Universal Robots URScript: etalement.script

# UR5 - Protocole etalement cosmetique
# Genere automatiquement par ur5_etalement.py
# IMPORTANT : calibrer ROBOT_X_ORIGIN, ROBOT_Y_ORIGIN, ROBOT_Z_SURFACE avant execution
#
# === RECETTE DE REPRODUCTION ===
# Ce bloc enonce ce qui a produit ce fichier. Il ne porte pas de date :
# une date rendrait l export non reproductible, et git la porte deja.
# cycles : 6
#   cycle 1 : type=circular waypoints=200   label=Cycle 1 - Circulaire (UI)
#   cycle 2 : type=circular waypoints=200   label=Cycle 2 - Circulaire (UI)
#   cycle 3 : type=circular waypoints=200   label=Cycle 3 - Circulaire (UI)
#   cycle 4 : type=linear   waypoints=14    label=Cycle 4 - Triangulé (0deg)
#   cycle 5 : type=linear   waypoints=14    label=Cycle 5 - Triangulé (90deg)
#   cycle 6 : type=linear   waypoints=14    label=Cycle 6 - Triangulé (0deg)
# empreinte des reglages : 44136fa
#
# === PINCE 2F-85 : AUCUN ACTIONNEMENT ===
# Ce programme n a pas de commande de pince. La 2F-85 est un support
# passif pour le doigt silicone ; seule sa longueur (TCP_GRIPPER_Z=145 mm)
# entre dans set_tcp(). Aucun rq_activate / rq_* / RS485 outil / set_payload.
# Erreur PolyScope "wait for activation completed" au chargement = URCap
# Robotiq Grippers de l INSTALLATION du robot (auto-activation BeforeStart),
# pas ce fichier. Corriger sur le robot : Installation > URCaps/Gripper >
# desactiver l auto-activation, ou retirer le URCap, ou charger sur une
# installation sans pince.
#

# --- Ancre de la zone d'etalement ---
global P_REF = p[-0.011, 0.6, 0.05, 3.14159, 0.0, 0.0]

# --- Vitesses (m/s) par phase ---
# Note : URSCRIPT_MAX_TCP_SPEED (limite PolyScope, 0.25 m/s) n'est pas
# emis ici ; il est applique par le controleur. La vitesse de transit
# est inlinee directement sur les movel de transit.
global URSCRIPT_CONTACT_V = 0.0500  #sym:URSCRIPT_CONTACT_V
global URSCRIPT_RECONTACT_V = 0.0100  #sym:URSCRIPT_RECONTACT_V
global V_CIRC = 0.0360  #sym:CIRC_SPEED
global V_RECT = 0.0800  #sym:LIN_SPEED

# --- Accelerations (m/s^2) par phase ---
global URSCRIPT_ACCEL = 0.8  #sym:URSCRIPT_ACCEL
global A_INIT = 1.2  #sym:A_INIT

# --- Facteurs multiplicateurs globaux ---
global SPEED_FACTOR = 1.0
global ACCEL_FACTOR = 1.0
global URSCRIPT_BLEND = 0.002  #sym:URSCRIPT_BLEND

# --- Sondage de surface : 1 point en Z (sondage 3 points DESACTIVE, voir bloc commente) ---
global PROBE_FORCE_THR    = 4.0
global PROBE_DESCENT_V    = 0.0040
global PROBE_ACCEL        = 0.05
global PROBE_MAX_TRAVEL   = 0.15
global NOMINAL_FRAME = p[-0.011000, 0.592930, 0.050004, 3.141576, 0.000000, 0.000000]
global MEAS_FRAME = p[-0.011000, 0.592930, 0.050004, 3.141576, 0.000000, 0.000000]
global contact_found = False
global contact_pose = p[0,0,0,0,0,0]

# --- Sondage Z (1 point) : trouve le plan de la plaque par contact force ---
# Depart = pose courante (operateur jogge le doigt juste au-dessus du
# plateau). Descente en -Z (base) jusqu au contact ; le Z touche devient
# la reference de TOUS les cycles 1 a 6 via MEAS_FRAME.
def probe_surface_z():
  textmsg(">>> Sondage Z : 1 point (recherche du plateau)")
  start_pose = get_actual_tcp_pose()
  zero_ftsensor()
  sleep(0.2)
  # CB3 (PolyScope 3.x) : descente surveillee dans le thread principal
  # (speedl non bloquant + lecture force + stopl). Pas de thread (stopl/
  # movel interdits dans un thread). get_tcp_force() lu en entier, norme
  # calculee a la main (pas de slice [0:3], absent du parser CB3).
  f_norm = 0.0
  travel = 0.0
  while f_norm <= PROBE_FORCE_THR and travel < PROBE_MAX_TRAVEL:
    speedl([0, 0, -PROBE_DESCENT_V, 0, 0, 0], PROBE_ACCEL, 0.05)
    F_tcp = get_tcp_force()
    f_norm = sqrt(F_tcp[0]*F_tcp[0] + F_tcp[1]*F_tcp[1] + F_tcp[2]*F_tcp[2])
    cur = get_actual_tcp_pose()
    travel = start_pose[2] - cur[2]
  end
  stopl(2.0)
  if f_norm <= PROBE_FORCE_THR:
    popup("Sondage Z echoue - aucun contact", "Rapprocher le doigt du plateau puis relancer", error=True)
    halt
  end
  touch = get_actual_tcp_pose()
  # Reference Z des cycles : repere nominal translate en Z jusqu au plan
  # touche. Orientation/XY restent nominaux (1 point ne mesure pas
  # l inclinaison -> rework futur). apply_correction decale chaque
  # waypoint du meme dz ; force_mode(MEAS_FRAME) regule les 6 N en Z.
  MEAS_FRAME = p[NOMINAL_FRAME[0], NOMINAL_FRAME[1], touch[2], NOMINAL_FRAME[3], NOMINAL_FRAME[4], NOMINAL_FRAME[5]]
  textmsg("Plateau detecte, Z (m) = ", touch[2])
end

def apply_correction(p_world):
  return pose_trans(MEAS_FRAME, pose_trans(pose_inv(NOMINAL_FRAME), p_world))
end

def cycle_1():
  # --- Cycle 1 - Circulaire (UI) ---
  movel(apply_correction(p[-0.017788, 0.586142, 0.060004, 3.141576, 0.000000, 0.000000]), a=URSCRIPT_ACCEL*ACCEL_FACTOR, v=0.2500*SPEED_FACTOR)
  sleep(0.2)
  zero_ftsensor()
  sleep(0.2)
  force_mode(MEAS_FRAME, [0, 0, 1, 0, 0, 0], [0, 0, -6.0, 0, 0, 0], 2, [0.008, 0.008, 0.04, 0.35, 0.35, 0.35])
  movel(apply_correction(p[-0.017788, 0.586142, 0.045004, 3.141576, 0.000000, 0.000000]), a=URSCRIPT_ACCEL*ACCEL_FACTOR, v=URSCRIPT_RECONTACT_V*SPEED_FACTOR)
  movel(apply_correction(p[-0.017788, 0.586142, 0.050004, 3.141576, 0.000000, 0.000000]), a=URSCRIPT_ACCEL*ACCEL_FACTOR, v=V_CIRC*SPEED_FACTOR, r=URSCRIPT_BLEND)
  movel(apply_correction(p[-0.011098, 0.583533, 0.050004, 3.141576, 0.000000, 0.000000]), a=URSCRIPT_ACCEL*ACCEL_FACTOR, v=V_CIRC*SPEED_FACTOR, r=URSCRIPT_BLEND)
  movel(apply_correction(p[-0.004916, 0.587048, 0.050004, 3.141576, 0.000000, 0.000000]), a=URSCRIPT_ACCEL*ACCEL_FACTOR, v=V_CIRC*SPEED_FACTOR, r=URSCRIPT_BLEND)
  movel(apply_correction(p[-0.005086, 0.594004, 0.050004, 3.141576, 0.000000, 0.000000]), a=URSCRIPT_ACCEL*ACCEL_FACTOR, v=V_CIRC*SPEED_FACTOR, r=URSCRIPT_BLEND)
  movel(apply_correction(p[-0.011712, 0.596025, 0.050004, 3.141576, 0.000000, 0.000000]), a=URSCRIPT_ACCEL*ACCEL_FACTOR, v=V_CIRC*SPEED_FACTOR, r=URSCRIPT_BLEND)
  movel(apply_correction(p[-0.016472, 0.590781, 0.050004, 3.141576, 0.000000, 0.000000]), a=URSCRIPT_ACCEL*ACCEL_FACTOR, v=V_CIRC*SPEED_FACTOR, r=URSCRIPT_BLEND)
  movel(apply_correction(p[-0.015164, 0.583730, 0.050004, 3.141576, 0.000000, 0.000000]), a=URSCRIPT_ACCEL*ACCEL_FACTOR, v=V_CIRC*SPEED_FACTOR, r=URSCRIPT_BLEND)
  movel(apply_correction(p[-0.009065, 0.579930, 0.050004, 3.141576, 0.000000, 0.000000]), a=URSCRIPT_ACCEL*ACCEL_FACTOR, v=V_CIRC*SPEED_FACTOR, r=URSCRIPT_BLEND)
  movel(apply_correction(p[-0.002264, 0.582086, 0.050004, 3.141576, 0.000000, 0.000000]), a=URSCRIPT_ACCEL*ACCEL_FACTOR, v=V_CIRC*SPEED_FACTOR, r=URSCRIPT_BLEND)
  movel(apply_correction(p[-0.000623, 0.588885, 0.050004, 3.141576, 0.000000, 0.000000]), a=URSCRIPT_ACCEL*ACCEL_FACTOR, v=V_CIRC*SPEED_FACTOR, r=URSCRIPT_BLEND)
  movel(apply_correction(p[-0.006418, 0.592643, 0.050004, 3.141576, 0.000000, 0.000000]), a=URSCRIPT_ACCEL*ACCEL_FACTOR, v=V_CIRC*SPEED_FACTOR, r=URSCRIPT_BLEND)
  movel(apply_correction(p[-0.012226, 0.588648, 0.050004, 3.141576, 0.000000, 0.000000]), a=URSCRIPT_ACCEL*ACCEL_FACTOR, v=V_CIRC*SPEED_FACTOR, r=URSCRIPT_BLEND)
  movel(apply_correction(p[-0.012291, 0.581489, 0.050004, 3.141576, 0.000000, 0.000000]), a=URSCRIPT_ACCEL*ACCEL_FACTOR, v=V_CIRC*SPEED_FACTOR, r=URSCRIPT_BLEND)
  movel(apply_correction(p[-0.006988, 0.576638, 0.050004, 3.141576, 0.000000, 0.000000]), a=URSCRIPT_ACCEL*ACCEL_FACTOR, v=V_CIRC*SPEED_FACTOR, r=URSCRIPT_BLEND)
  movel(apply_correction(p[0.000125, 0.577386, 0.050004, 3.141576, 0.000000, 0.000000]), a=URSCRIPT_ACCEL*ACCEL_FACTOR, v=V_CIRC*SPEED_FACTOR, r=URSCRIPT_BLEND)
  movel(apply_correction(p[0.003408, 0.583603, 0.050004, 3.141576, 0.000000, 0.000000]), a=URSCRIPT_ACCEL*ACCEL_FACTOR, v=V_CIRC*SPEED_FACTOR, r=URSCRIPT_BLEND)
  movel(apply_correction(p[-0.001104, 0.588825, 0.050004, 3.141576, 0.000000, 0.000000]), a=URSCRIPT_ACCEL*ACCEL_FACTOR, v=V_CIRC*SPEED_FACTOR, r=URSCRIPT_BLEND)
  movel(apply_correction(p[-0.007670, 0.586361, 0.050004, 3.141576, 0.000000, 0.000000]), a=URSCRIPT_ACCEL*ACCEL_FACTOR, v=V_CIRC*SPEED_FACTOR, r=URSCRIPT_BLEND)
  movel(apply_correction(p[-0.009144, 0.579371, 0.050004, 3.141576, 0.000000, 0.000000]), a=URSCRIPT_ACCEL*ACCEL_FACTOR, v=V_CIRC*SPEED_FACTOR, r=URSCRIPT_BLEND)
  movel(apply_correction(p[-0.004813, 0.573634, 0.050004, 3.141576, 0.000000, 0.000000]), a=URSCRIPT_ACCEL*ACCEL_FACTOR, v=V_CIRC*SPEED_FACTOR, r=URSCRIPT_BLEND)
  movel(apply_correction(p[0.002324, 0.572985, 0.050004, 3.141576, 0.000000, 0.000000]), a=URSCRIPT_ACCEL*ACCEL_FACTOR, v=V_CIRC*SPEED_FACTOR, r=URSCRIPT_BLEND)
  movel(apply_correction(p[0.006999, 0.578286, 0.050004, 3.141576, 0.000000, 0.000000]), a=URSCRIPT_ACCEL*ACCEL_FACTOR, v=V_CIRC*SPEED_FACTOR, r=URSCRIPT_BLEND)
  movel(apply_correction(p[0.004110, 0.584567, 0.050004, 3.141576, 0.000000, 0.000000]), a=URSCRIPT_ACCEL*ACCEL_FACTOR, v=V_CIRC*SPEED_FACTOR, r=URSCRIPT_BLEND)
  movel(apply_correction(p[-0.002829, 0.583846, 0.050004, 3.141576, 0.000000, 0.000000]), a=URSCRIPT_ACCEL*ACCEL_FACTOR, v=V_CIRC*SPEED_FACTOR, r=URSCRIPT_BLEND)
  movel(apply_correction(p[-0.005691, 0.577324, 0.050004, 3.141576, 0.000000, 0.000000]), a=URSCRIPT_ACCEL*ACCEL_FACTOR, v=V_CIRC*SPEED_FACTOR, r=URSCRIPT_BLEND)
  movel(apply_correction(p[-0.002490, 0.570894, 0.050004, 3.141576, 0.000000, 0.000000]), a=URSCRIPT_ACCEL*ACCEL_FACTOR, v=V_CIRC*SPEED_FACTOR, r=URSCRIPT_BLEND)
  movel(apply_correction(p[0.004406, 0.568905, 0.050004, 3.141576, 0.000000, 0.000000]), a=URSCRIPT_ACCEL*ACCEL_FACTOR, v=V_CIRC*SPEED_FACTOR, r=URSCRIPT_BLEND)
  movel(apply_correction(p[0.010171, 0.573044, 0.050004, 3.141576, 0.000000, 0.000000]), a=URSCRIPT_ACCEL*ACCEL_FACTOR, v=V_CIRC*SPEED_FACTOR, r=URSCRIPT_BLEND)
  movel(apply_correction(p[0.009098, 0.579900, 0.050004, 3.141576, 0.000000, 0.000000]), a=URSCRIPT_ACCEL*ACCEL_FACTOR, v=V_CIRC*SPEED_FACTOR, r=URSCRIPT_BLEND)
  movel(apply_correction(p[0.002251, 0.581029, 0.050004, 3.141576, 0.000000, 0.000000]), a=URSCRIPT_ACCEL*ACCEL_FACTOR, v=V_CIRC*SPEED_FACTOR, r=URSCRIPT_BLEND)
  movel(apply_correction(p[-0.001925, 0.575290, 0.050004, 3.141576, 0.000000, 0.000000]), a=URSCRIPT_ACCEL*ACCEL_FACTOR, v=V_CIRC*SPEED_FACTOR, r=URSCRIPT_BLEND)
  movel(apply_correction(p[0.000027, 0.568386, 0.050004, 3.141576, 0.000000, 0.000000]), a=URSCRIPT_ACCEL*ACCEL_FACTOR, v=V_CIRC*SPEED_FACTOR, r=URSCRIPT_BLEND)
  movel(apply_correction(p[0.006439, 0.565146, 0.050005, 3.141576, 0.000000, 0.000000]), a=URSCRIPT_ACCEL*ACCEL_FACTOR, v=V_CIRC*SPEED_FACTOR, r=URSCRIPT_BLEND)
  movel(apply_correction(p[0.012978, 0.567972, 0.050004, 3.141576, 0.000000, 0.000000]), a=URSCRIPT_ACCEL*ACCEL_FACTOR, v=V_CIRC*SPEED_FACTOR, r=URSCRIPT_BLEND)
  movel(apply_correction(p[0.013753, 0.574903, 0.050004, 3.141576, 0.000000, 0.000000]), a=URSCRIPT_ACCEL*ACCEL_FACTOR, v=V_CIRC*SPEED_FACTOR, r=URSCRIPT_BLEND)
  movel(apply_correction(p[0.007496, 0.577845, 0.050004, 3.141576, 0.000000, 0.000000]), a=URSCRIPT_ACCEL*ACCEL_FACTOR, v=V_CIRC*SPEED_FACTOR, r=URSCRIPT_BLEND)
  movel(apply_correction(p[0.002166, 0.573206, 0.050004, 3.141576, 0.000000, 0.000000]), a=URSCRIPT_ACCEL*ACCEL_FACTOR, v=V_CIRC*SPEED_FACTOR, r=URSCRIPT_BLEND)
  movel(apply_correction(p[0.002775, 0.566066, 0.050004, 3.141576, 0.000000, 0.000000]), a=URSCRIPT_ACCEL*ACCEL_FACTOR, v=V_CIRC*SPEED_FACTOR, r=URSCRIPT_BLEND)
  movel(apply_correction(p[0.008487, 0.561706, 0.050005, 3.141576, 0.000000, 0.000000]), a=URSCRIPT_ACCEL*ACCEL_FACTOR, v=V_CIRC*SPEED_FACTOR, r=URSCRIPT_BLEND)
  movel(apply_correction(p[0.015475, 0.563167, 0.050005, 3.141576, 0.000000, 0.000000]), a=URSCRIPT_ACCEL*ACCEL_FACTOR, v=V_CIRC*SPEED_FACTOR, r=URSCRIPT_BLEND)
  movel(apply_correction(p[0.017743, 0.569730, 0.050004, 3.141576, 0.000000, 0.000000]), a=URSCRIPT_ACCEL*ACCEL_FACTOR, v=V_CIRC*SPEED_FACTOR, r=URSCRIPT_BLEND)
  movel(apply_correction(p[0.012260, 0.573881, 0.050004, 3.141576, 0.000000, 0.000000]), a=URSCRIPT_ACCEL*ACCEL_FACTOR, v=V_CIRC*SPEED_FACTOR, r=URSCRIPT_BLEND)
  movel(apply_correction(p[0.005935, 0.570677, 0.050004, 3.141576, 0.000000, 0.000000]), a=URSCRIPT_ACCEL*ACCEL_FACTOR, v=V_CIRC*SPEED_FACTOR, r=URSCRIPT_BLEND)
  movel(apply_correction(p[0.004428, 0.563644, 0.050005, 3.141576, 0.000000, 0.000000]), a=URSCRIPT_ACCEL*ACCEL_FACTOR, v=V_CIRC*SPEED_FACTOR, r=URSCRIPT_BLEND)
  movel(apply_correction(p[0.008552, 0.557768, 0.050005, 3.141576, 0.000000, 0.000000]), a=URSCRIPT_ACCEL*ACCEL_FACTOR, v=V_CIRC*SPEED_FACTOR, r=URSCRIPT_BLEND)
  movel(apply_correction(p[0.015598, 0.557554, 0.050005, 3.141576, 0.000000, 0.000000]), a=URSCRIPT_ACCEL*ACCEL_FACTOR, v=V_CIRC*SPEED_FACTOR, r=URSCRIPT_BLEND)
  movel(apply_correction(p[0.018398, 0.563819, 0.050005, 3.141576, 0.000000, 0.000000]), a=URSCRIPT_ACCEL*ACCEL_FACTOR, v=V_CIRC*SPEED_FACTOR, r=URSCRIPT_BLEND)
  movel(apply_correction(p[0.013349, 0.568656, 0.050004, 3.141576, 0.000000, 0.000000]), a=URSCRIPT_ACCEL*ACCEL_FACTOR, v=V_CIRC*SPEED_FACTOR, r=URSCRIPT_BLEND)
  movel(apply_correction(p[0.006365, 0.567164, 0.050004, 3.141576, 0.000000, 0.000000]), a=URSCRIPT_ACCEL*ACCEL_FACTOR, v=V_CIRC*SPEED_FACTOR, r=URSCRIPT_BLEND)
  movel(apply_correction(p[0.002726, 0.560986, 0.050005, 3.141576, 0.000000, 0.000000]), a=URSCRIPT_ACCEL*ACCEL_FACTOR, v=V_CIRC*SPEED_FACTOR, r=URSCRIPT_BLEND)
  movel(apply_correction(p[0.004975, 0.554229, 0.050005, 3.141576, 0.000000, 0.000000]), a=URSCRIPT_ACCEL*ACCEL_FACTOR, v=V_CIRC*SPEED_FACTOR, r=URSCRIPT_BLEND)
  movel(apply_correction(p[0.011813, 0.552992, 0.050005, 3.141576, 0.000000, 0.000000]), a=URSCRIPT_ACCEL*ACCEL_FACTOR, v=V_CIRC*SPEED_FACTOR, r=URSCRIPT_BLEND)
  movel(apply_correction(p[0.015059, 0.559096, 0.050005, 3.141576, 0.000000, 0.000000]), a=URSCRIPT_ACCEL*ACCEL_FACTOR, v=V_CIRC*SPEED_FACTOR, r=URSCRIPT_BLEND)
  movel(apply_correction(p[0.011046, 0.564958, 0.050005, 3.141576, 0.000000, 0.000000]), a=URSCRIPT_ACCEL*ACCEL_FACTOR, v=V_CIRC*SPEED_FACTOR, r=URSCRIPT_BLEND)
  movel(apply_correction(p[0.003896, 0.565651, 0.050004, 3.141576, 0.000000, 0.000000]), a=URSCRIPT_ACCEL*ACCEL_FACTOR, v=V_CIRC*SPEED_FACTOR, r=URSCRIPT_BLEND)
  movel(apply_correction(p[-0.001449, 0.560893, 0.050005, 3.141576, 0.000000, 0.000000]), a=URSCRIPT_ACCEL*ACCEL_FACTOR, v=V_CIRC*SPEED_FACTOR, r=URSCRIPT_BLEND)
  movel(apply_correction(p[-0.000730, 0.553895, 0.050005, 3.141576, 0.000000, 0.000000]), a=URSCRIPT_ACCEL*ACCEL_FACTOR, v=V_CIRC*SPEED_FACTOR, r=URSCRIPT_BLEND)
  movel(apply_correction(p[0.005938, 0.552136, 0.050005, 3.141576, 0.000000, 0.000000]), a=URSCRIPT_ACCEL*ACCEL_FACTOR, v=V_CIRC*SPEED_FACTOR, r=URSCRIPT_BLEND)
  movel(apply_correction(p[0.010014, 0.557869, 0.050005, 3.141576, 0.000000, 0.000000]), a=URSCRIPT_ACCEL*ACCEL_FACTOR, v=V_CIRC*SPEED_FACTOR, r=URSCRIPT_BLEND)
  movel(apply_correction(p[0.007718, 0.564641, 0.050005, 3.141576, 0.000000, 0.000000]), a=URSCRIPT_ACCEL*ACCEL_FACTOR, v=V_CIRC*SPEED_FACTOR, r=URSCRIPT_BLEND)
  movel(apply_correction(p[0.001166, 0.567570, 0.050004, 3.141576, 0.000000, 0.000000]), a=URSCRIPT_ACCEL*ACCEL_FACTOR, v=V_CIRC*SPEED_FACTOR, r=URSCRIPT_BLEND)
  movel(apply_correction(p[-0.005246, 0.564498, 0.050005, 3.141576, 0.000000, 0.000000]), a=URSCRIPT_ACCEL*ACCEL_FACTOR, v=V_CIRC*SPEED_FACTOR, r=URSCRIPT_BLEND)
  movel(apply_correction(p[-0.005654, 0.557540, 0.050005, 3.141576, 0.000000, 0.000000]), a=URSCRIPT_ACCEL*ACCEL_FACTOR, v=V_CIRC*SPEED_FACTOR, r=URSCRIPT_BLEND)
  movel(apply_correction(p[0.000763, 0.554955, 0.050005, 3.141576, 0.000000, 0.000000]), a=URSCRIPT_ACCEL*ACCEL_FACTOR, v=V_CIRC*SPEED_FACTOR, r=URSCRIPT_BLEND)
  movel(apply_correction(p[0.005879, 0.559839, 0.050005, 3.141576, 0.000000, 0.000000]), a=URSCRIPT_ACCEL*ACCEL_FACTOR, v=V_CIRC*SPEED_FACTOR, r=URSCRIPT_BLEND)
  movel(apply_correction(p[0.004993, 0.566952, 0.050004, 3.141576, 0.000000, 0.000000]), a=URSCRIPT_ACCEL*ACCEL_FACTOR, v=V_CIRC*SPEED_FACTOR, r=URSCRIPT_BLEND)
  movel(apply_correction(p[-0.000876, 0.571099, 0.050004, 3.141576, 0.000000, 0.000000]), a=URSCRIPT_ACCEL*ACCEL_FACTOR, v=V_CIRC*SPEED_FACTOR, r=URSCRIPT_BLEND)
  movel(apply_correction(p[-0.007807, 0.569384, 0.050004, 3.141576, 0.000000, 0.000000]), a=URSCRIPT_ACCEL*ACCEL_FACTOR, v=V_CIRC*SPEED_FACTOR, r=URSCRIPT_BLEND)
  movel(apply_correction(p[-0.009985, 0.562724, 0.050005, 3.141576, 0.000000, 0.000000]), a=URSCRIPT_ACCEL*ACCEL_FACTOR, v=V_CIRC*SPEED_FACTOR, r=URSCRIPT_BLEND)
  movel(apply_correction(p[-0.004550, 0.558471, 0.050005, 3.141576, 0.000000, 0.000000]), a=URSCRIPT_ACCEL*ACCEL_FACTOR, v=V_CIRC*SPEED_FACTOR, r=URSCRIPT_BLEND)
  movel(apply_correction(p[0.001532, 0.562013, 0.050005, 3.141576, 0.000000, 0.000000]), a=URSCRIPT_ACCEL*ACCEL_FACTOR, v=V_CIRC*SPEED_FACTOR, r=URSCRIPT_BLEND)
  movel(apply_correction(p[0.002038, 0.569150, 0.050004, 3.141576, 0.000000, 0.000000]), a=URSCRIPT_ACCEL*ACCEL_FACTOR, v=V_CIRC*SPEED_FACTOR, r=URSCRIPT_BLEND)
  movel(apply_correction(p[-0.002979, 0.574298, 0.050004, 3.141576, 0.000000, 0.000000]), a=URSCRIPT_ACCEL*ACCEL_FACTOR, v=V_CIRC*SPEED_FACTOR, r=URSCRIPT_BLEND)
  movel(apply_correction(p[-0.010128, 0.573991, 0.050004, 3.141576, 0.000000, 0.000000]), a=URSCRIPT_ACCEL*ACCEL_FACTOR, v=V_CIRC*SPEED_FACTOR, r=URSCRIPT_BLEND)
  movel(apply_correction(p[-0.013879, 0.568031, 0.050004, 3.141576, 0.000000, 0.000000]), a=URSCRIPT_ACCEL*ACCEL_FACTOR, v=V_CIRC*SPEED_FACTOR, r=URSCRIPT_BLEND)
  movel(apply_correction(p[-0.009845, 0.562427, 0.050005, 3.141576, 0.000000, 0.000000]), a=URSCRIPT_ACCEL*ACCEL_FACTOR, v=V_CIRC*SPEED_FACTOR, r=URSCRIPT_BLEND)
  movel(apply_correction(p[-0.003119, 0.564364, 0.050005, 3.141576, 0.000000, 0.000000]), a=URSCRIPT_ACCEL*ACCEL_FACTOR, v=V_CIRC*SPEED_FACTOR, r=URSCRIPT_BLEND)
  movel(apply_correction(p[-0.001202, 0.571240, 0.050004, 3.141576, 0.000000, 0.000000]), a=URSCRIPT_ACCEL*ACCEL_FACTOR, v=V_CIRC*SPEED_FACTOR, r=URSCRIPT_BLEND)
  movel(apply_correction(p[-0.005195, 0.577216, 0.050004, 3.141576, 0.000000, 0.000000]), a=URSCRIPT_ACCEL*ACCEL_FACTOR, v=V_CIRC*SPEED_FACTOR, r=URSCRIPT_BLEND)
  movel(apply_correction(p[-0.012283, 0.578294, 0.050004, 3.141576, 0.000000, 0.000000]), a=URSCRIPT_ACCEL*ACCEL_FACTOR, v=V_CIRC*SPEED_FACTOR, r=URSCRIPT_BLEND)
  movel(apply_correction(p[-0.017334, 0.573336, 0.050004, 3.141576, 0.000000, 0.000000]), a=URSCRIPT_ACCEL*ACCEL_FACTOR, v=V_CIRC*SPEED_FACTOR, r=URSCRIPT_BLEND)
  movel(apply_correction(p[-0.015002, 0.566819, 0.050004, 3.141576, 0.000000, 0.000000]), a=URSCRIPT_ACCEL*ACCEL_FACTOR, v=V_CIRC*SPEED_FACTOR, r=URSCRIPT_BLEND)
  movel(apply_correction(p[-0.008039, 0.566966, 0.050004, 3.141576, 0.000000, 0.000000]), a=URSCRIPT_ACCEL*ACCEL_FACTOR, v=V_CIRC*SPEED_FACTOR, r=URSCRIPT_BLEND)
  movel(apply_correction(p[-0.004752, 0.573277, 0.050004, 3.141576, 0.000000, 0.000000]), a=URSCRIPT_ACCEL*ACCEL_FACTOR, v=V_CIRC*SPEED_FACTOR, r=URSCRIPT_BLEND)
  movel(apply_correction(p[-0.007574, 0.579880, 0.050004, 3.141576, 0.000000, 0.000000]), a=URSCRIPT_ACCEL*ACCEL_FACTOR, v=V_CIRC*SPEED_FACTOR, r=URSCRIPT_BLEND)
  movel(apply_correction(p[-0.014343, 0.582272, 0.050004, 3.141576, 0.000000, 0.000000]), a=URSCRIPT_ACCEL*ACCEL_FACTOR, v=V_CIRC*SPEED_FACTOR, r=URSCRIPT_BLEND)
  movel(apply_correction(p[-0.020386, 0.578533, 0.050004, 3.141576, 0.000000, 0.000000]), a=URSCRIPT_ACCEL*ACCEL_FACTOR, v=V_CIRC*SPEED_FACTOR, r=URSCRIPT_BLEND)
  movel(apply_correction(p[-0.019895, 0.571600, 0.050004, 3.141576, 0.000000, 0.000000]), a=URSCRIPT_ACCEL*ACCEL_FACTOR, v=V_CIRC*SPEED_FACTOR, r=URSCRIPT_BLEND)
  movel(apply_correction(p[-0.013179, 0.569890, 0.050004, 3.141576, 0.000000, 0.000000]), a=URSCRIPT_ACCEL*ACCEL_FACTOR, v=V_CIRC*SPEED_FACTOR, r=URSCRIPT_BLEND)
  movel(apply_correction(p[-0.008631, 0.575334, 0.050004, 3.141576, 0.000000, 0.000000]), a=URSCRIPT_ACCEL*ACCEL_FACTOR, v=V_CIRC*SPEED_FACTOR, r=URSCRIPT_BLEND)
  movel(apply_correction(p[-0.010345, 0.582287, 0.050004, 3.141576, 0.000000, 0.000000]), a=URSCRIPT_ACCEL*ACCEL_FACTOR, v=V_CIRC*SPEED_FACTOR, r=URSCRIPT_BLEND)
  movel(apply_correction(p[-0.016696, 0.585620, 0.050004, 3.141576, 0.000000, 0.000000]), a=URSCRIPT_ACCEL*ACCEL_FACTOR, v=V_CIRC*SPEED_FACTOR, r=URSCRIPT_BLEND)
  movel(apply_correction(p[-0.023362, 0.583056, 0.050004, 3.141576, 0.000000, 0.000000]), a=URSCRIPT_ACCEL*ACCEL_FACTOR, v=V_CIRC*SPEED_FACTOR, r=URSCRIPT_BLEND)
  movel(apply_correction(p[-0.025236, 0.576243, 0.050004, 3.141576, 0.000000, 0.000000]), a=URSCRIPT_ACCEL*ACCEL_FACTOR, v=V_CIRC*SPEED_FACTOR, r=URSCRIPT_BLEND)
  movel(apply_correction(p[-0.020034, 0.571653, 0.050004, 3.141576, 0.000000, 0.000000]), a=URSCRIPT_ACCEL*ACCEL_FACTOR, v=V_CIRC*SPEED_FACTOR, r=URSCRIPT_BLEND)
  movel(apply_correction(p[-0.014038, 0.575090, 0.050004, 3.141576, 0.000000, 0.000000]), a=URSCRIPT_ACCEL*ACCEL_FACTOR, v=V_CIRC*SPEED_FACTOR, r=URSCRIPT_BLEND)
  movel(apply_correction(p[-0.014738, 0.582089, 0.050004, 3.141576, 0.000000, 0.000000]), a=URSCRIPT_ACCEL*ACCEL_FACTOR, v=V_CIRC*SPEED_FACTOR, r=URSCRIPT_BLEND)
  movel(apply_correction(p[-0.020976, 0.585534, 0.050004, 3.141576, 0.000000, 0.000000]), a=URSCRIPT_ACCEL*ACCEL_FACTOR, v=V_CIRC*SPEED_FACTOR, r=URSCRIPT_BLEND)
  movel(apply_correction(p[-0.027687, 0.583050, 0.050004, 3.141576, 0.000000, 0.000000]), a=URSCRIPT_ACCEL*ACCEL_FACTOR, v=V_CIRC*SPEED_FACTOR, r=URSCRIPT_BLEND)
  movel(apply_correction(p[-0.030305, 0.576399, 0.050004, 3.141576, 0.000000, 0.000000]), a=URSCRIPT_ACCEL*ACCEL_FACTOR, v=V_CIRC*SPEED_FACTOR, r=URSCRIPT_BLEND)
  movel(apply_correction(p[-0.026697, 0.570296, 0.050004, 3.141576, 0.000000, 0.000000]), a=URSCRIPT_ACCEL*ACCEL_FACTOR, v=V_CIRC*SPEED_FACTOR, r=URSCRIPT_BLEND)
  movel(apply_correction(p[-0.019718, 0.570534, 0.050004, 3.141576, 0.000000, 0.000000]), a=URSCRIPT_ACCEL*ACCEL_FACTOR, v=V_CIRC*SPEED_FACTOR, r=URSCRIPT_BLEND)
  movel(apply_correction(p[-0.017643, 0.577142, 0.050004, 3.141576, 0.000000, 0.000000]), a=URSCRIPT_ACCEL*ACCEL_FACTOR, v=V_CIRC*SPEED_FACTOR, r=URSCRIPT_BLEND)
  movel(apply_correction(p[-0.023092, 0.581572, 0.050004, 3.141576, 0.000000, 0.000000]), a=URSCRIPT_ACCEL*ACCEL_FACTOR, v=V_CIRC*SPEED_FACTOR, r=URSCRIPT_BLEND)
  movel(apply_correction(p[-0.029871, 0.579381, 0.050004, 3.141576, 0.000000, 0.000000]), a=URSCRIPT_ACCEL*ACCEL_FACTOR, v=V_CIRC*SPEED_FACTOR, r=URSCRIPT_BLEND)
  movel(apply_correction(p[-0.032536, 0.572708, 0.050004, 3.141576, 0.000000, 0.000000]), a=URSCRIPT_ACCEL*ACCEL_FACTOR, v=V_CIRC*SPEED_FACTOR, r=URSCRIPT_BLEND)
  movel(apply_correction(p[-0.029339, 0.566277, 0.050004, 3.141576, 0.000000, 0.000000]), a=URSCRIPT_ACCEL*ACCEL_FACTOR, v=V_CIRC*SPEED_FACTOR, r=URSCRIPT_BLEND)
  movel(apply_correction(p[-0.022399, 0.564726, 0.050005, 3.141576, 0.000000, 0.000000]), a=URSCRIPT_ACCEL*ACCEL_FACTOR, v=V_CIRC*SPEED_FACTOR, r=URSCRIPT_BLEND)
  movel(apply_correction(p[-0.017535, 0.569747, 0.050004, 3.141576, 0.000000, 0.000000]), a=URSCRIPT_ACCEL*ACCEL_FACTOR, v=V_CIRC*SPEED_FACTOR, r=URSCRIPT_BLEND)
  movel(apply_correction(p[-0.020477, 0.575989, 0.050004, 3.141576, 0.000000, 0.000000]), a=URSCRIPT_ACCEL*ACCEL_FACTOR, v=V_CIRC*SPEED_FACTOR, r=URSCRIPT_BLEND)
  movel(apply_correction(p[-0.027450, 0.575397, 0.050004, 3.141576, 0.000000, 0.000000]), a=URSCRIPT_ACCEL*ACCEL_FACTOR, v=V_CIRC*SPEED_FACTOR, r=URSCRIPT_BLEND)
  movel(apply_correction(p[-0.030496, 0.568956, 0.050004, 3.141576, 0.000000, 0.000000]), a=URSCRIPT_ACCEL*ACCEL_FACTOR, v=V_CIRC*SPEED_FACTOR, r=URSCRIPT_BLEND)
  movel(apply_correction(p[-0.027445, 0.562453, 0.050005, 3.141576, 0.000000, 0.000000]), a=URSCRIPT_ACCEL*ACCEL_FACTOR, v=V_CIRC*SPEED_FACTOR, r=URSCRIPT_BLEND)
  movel(apply_correction(p[-0.020600, 0.560297, 0.050005, 3.141576, 0.000000, 0.000000]), a=URSCRIPT_ACCEL*ACCEL_FACTOR, v=V_CIRC*SPEED_FACTOR, r=URSCRIPT_BLEND)
  movel(apply_correction(p[-0.014717, 0.564274, 0.050005, 3.141576, 0.000000, 0.000000]), a=URSCRIPT_ACCEL*ACCEL_FACTOR, v=V_CIRC*SPEED_FACTOR, r=URSCRIPT_BLEND)
  movel(apply_correction(p[-0.015552, 0.571170, 0.050004, 3.141576, 0.000000, 0.000000]), a=URSCRIPT_ACCEL*ACCEL_FACTOR, v=V_CIRC*SPEED_FACTOR, r=URSCRIPT_BLEND)
  movel(apply_correction(p[-0.022352, 0.572534, 0.050004, 3.141576, 0.000000, 0.000000]), a=URSCRIPT_ACCEL*ACCEL_FACTOR, v=V_CIRC*SPEED_FACTOR, r=URSCRIPT_BLEND)
  movel(apply_correction(p[-0.026686, 0.566919, 0.050004, 3.141576, 0.000000, 0.000000]), a=URSCRIPT_ACCEL*ACCEL_FACTOR, v=V_CIRC*SPEED_FACTOR, r=URSCRIPT_BLEND)
  movel(apply_correction(p[-0.024903, 0.559969, 0.050005, 3.141576, 0.000000, 0.000000]), a=URSCRIPT_ACCEL*ACCEL_FACTOR, v=V_CIRC*SPEED_FACTOR, r=URSCRIPT_BLEND)
  movel(apply_correction(p[-0.018568, 0.556581, 0.050005, 3.141576, 0.000000, 0.000000]), a=URSCRIPT_ACCEL*ACCEL_FACTOR, v=V_CIRC*SPEED_FACTOR, r=URSCRIPT_BLEND)
  movel(apply_correction(p[-0.011952, 0.559230, 0.050005, 3.141576, 0.000000, 0.000000]), a=URSCRIPT_ACCEL*ACCEL_FACTOR, v=V_CIRC*SPEED_FACTOR, r=URSCRIPT_BLEND)
  movel(apply_correction(p[-0.010947, 0.566137, 0.050004, 3.141576, 0.000000, 0.000000]), a=URSCRIPT_ACCEL*ACCEL_FACTOR, v=V_CIRC*SPEED_FACTOR, r=URSCRIPT_BLEND)
  movel(apply_correction(p[-0.017092, 0.569298, 0.050004, 3.141576, 0.000000, 0.000000]), a=URSCRIPT_ACCEL*ACCEL_FACTOR, v=V_CIRC*SPEED_FACTOR, r=URSCRIPT_BLEND)
  movel(apply_correction(p[-0.022556, 0.564825, 0.050005, 3.141576, 0.000000, 0.000000]), a=URSCRIPT_ACCEL*ACCEL_FACTOR, v=V_CIRC*SPEED_FACTOR, r=URSCRIPT_BLEND)
  movel(apply_correction(p[-0.022123, 0.557672, 0.050005, 3.141576, 0.000000, 0.000000]), a=URSCRIPT_ACCEL*ACCEL_FACTOR, v=V_CIRC*SPEED_FACTOR, r=URSCRIPT_BLEND)
  movel(apply_correction(p[-0.016514, 0.553178, 0.050005, 3.141576, 0.000000, 0.000000]), a=URSCRIPT_ACCEL*ACCEL_FACTOR, v=V_CIRC*SPEED_FACTOR, r=URSCRIPT_BLEND)
  movel(apply_correction(p[-0.009477, 0.554429, 0.050005, 3.141576, 0.000000, 0.000000]), a=URSCRIPT_ACCEL*ACCEL_FACTOR, v=V_CIRC*SPEED_FACTOR, r=URSCRIPT_BLEND)
  movel(apply_correction(p[-0.006757, 0.560900, 0.050005, 3.141576, 0.000000, 0.000000]), a=URSCRIPT_ACCEL*ACCEL_FACTOR, v=V_CIRC*SPEED_FACTOR, r=URSCRIPT_BLEND)
  movel(apply_correction(p[-0.011771, 0.565641, 0.050004, 3.141576, 0.000000, 0.000000]), a=URSCRIPT_ACCEL*ACCEL_FACTOR, v=V_CIRC*SPEED_FACTOR, r=URSCRIPT_BLEND)
  movel(apply_correction(p[-0.018106, 0.562599, 0.050005, 3.141576, 0.000000, 0.000000]), a=URSCRIPT_ACCEL*ACCEL_FACTOR, v=V_CIRC*SPEED_FACTOR, r=URSCRIPT_BLEND)
  movel(apply_correction(p[-0.019075, 0.555515, 0.050005, 3.141576, 0.000000, 0.000000]), a=URSCRIPT_ACCEL*ACCEL_FACTOR, v=V_CIRC*SPEED_FACTOR, r=URSCRIPT_BLEND)
  movel(apply_correction(p[-0.014379, 0.550076, 0.050005, 3.141576, 0.000000, 0.000000]), a=URSCRIPT_ACCEL*ACCEL_FACTOR, v=V_CIRC*SPEED_FACTOR, r=URSCRIPT_BLEND)
  movel(apply_correction(p[-0.007220, 0.549921, 0.050005, 3.141576, 0.000000, 0.000000]), a=URSCRIPT_ACCEL*ACCEL_FACTOR, v=V_CIRC*SPEED_FACTOR, r=URSCRIPT_BLEND)
  movel(apply_correction(p[-0.003008, 0.555581, 0.050005, 3.141576, 0.000000, 0.000000]), a=URSCRIPT_ACCEL*ACCEL_FACTOR, v=V_CIRC*SPEED_FACTOR, r=URSCRIPT_BLEND)
  movel(apply_correction(p[-0.006508, 0.561538, 0.050005, 3.141576, 0.000000, 0.000000]), a=URSCRIPT_ACCEL*ACCEL_FACTOR, v=V_CIRC*SPEED_FACTOR, r=URSCRIPT_BLEND)
  movel(apply_correction(p[-0.013362, 0.560174, 0.050005, 3.141576, 0.000000, 0.000000]), a=URSCRIPT_ACCEL*ACCEL_FACTOR, v=V_CIRC*SPEED_FACTOR, r=URSCRIPT_BLEND)
  movel(apply_correction(p[-0.015736, 0.553449, 0.050005, 3.141576, 0.000000, 0.000000]), a=URSCRIPT_ACCEL*ACCEL_FACTOR, v=V_CIRC*SPEED_FACTOR, r=URSCRIPT_BLEND)
  movel(apply_correction(p[-0.012114, 0.547244, 0.050005, 3.141576, 0.000000, 0.000000]), a=URSCRIPT_ACCEL*ACCEL_FACTOR, v=V_CIRC*SPEED_FACTOR, r=URSCRIPT_BLEND)
  movel(apply_correction(p[-0.005103, 0.545724, 0.050005, 3.141576, 0.000000, 0.000000]), a=URSCRIPT_ACCEL*ACCEL_FACTOR, v=V_CIRC*SPEED_FACTOR, r=URSCRIPT_BLEND)
  movel(apply_correction(p[0.000267, 0.550317, 0.050005, 3.141576, 0.000000, 0.000000]), a=URSCRIPT_ACCEL*ACCEL_FACTOR, v=V_CIRC*SPEED_FACTOR, r=URSCRIPT_BLEND)
  movel(apply_correction(p[-0.001550, 0.556944, 0.050005, 3.141576, 0.000000, 0.000000]), a=URSCRIPT_ACCEL*ACCEL_FACTOR, v=V_CIRC*SPEED_FACTOR, r=URSCRIPT_BLEND)
  movel(apply_correction(p[-0.008498, 0.557307, 0.050005, 3.141576, 0.000000, 0.000000]), a=URSCRIPT_ACCEL*ACCEL_FACTOR, v=V_CIRC*SPEED_FACTOR, r=URSCRIPT_BLEND)
  movel(apply_correction(p[-0.012498, 0.551407, 0.050005, 3.141576, 0.000000, 0.000000]), a=URSCRIPT_ACCEL*ACCEL_FACTOR, v=V_CIRC*SPEED_FACTOR, r=URSCRIPT_BLEND)
  movel(apply_correction(p[-0.010765, 0.544449, 0.050005, 3.141576, 0.000000, 0.000000]), a=URSCRIPT_ACCEL*ACCEL_FACTOR, v=V_CIRC*SPEED_FACTOR, r=URSCRIPT_BLEND)
  movel(apply_correction(p[-0.004471, 0.541100, 0.050005, 3.141576, 0.000000, 0.000000]), a=URSCRIPT_ACCEL*ACCEL_FACTOR, v=V_CIRC*SPEED_FACTOR, r=URSCRIPT_BLEND)
  movel(apply_correction(p[0.001548, 0.544594, 0.050005, 3.141576, 0.000000, 0.000000]), a=URSCRIPT_ACCEL*ACCEL_FACTOR, v=V_CIRC*SPEED_FACTOR, r=URSCRIPT_BLEND)
  movel(apply_correction(p[0.000165, 0.551320, 0.050005, 3.141576, 0.000000, 0.000000]), a=URSCRIPT_ACCEL*ACCEL_FACTOR, v=V_CIRC*SPEED_FACTOR, r=URSCRIPT_BLEND)
  movel(apply_correction(p[-0.006728, 0.552924, 0.050005, 3.141576, 0.000000, 0.000000]), a=URSCRIPT_ACCEL*ACCEL_FACTOR, v=V_CIRC*SPEED_FACTOR, r=URSCRIPT_BLEND)
  movel(apply_correction(p[-0.012333, 0.548421, 0.050005, 3.141576, 0.000000, 0.000000]), a=URSCRIPT_ACCEL*ACCEL_FACTOR, v=V_CIRC*SPEED_FACTOR, r=URSCRIPT_BLEND)
  movel(apply_correction(p[-0.012858, 0.541260, 0.050005, 3.141576, 0.000000, 0.000000]), a=URSCRIPT_ACCEL*ACCEL_FACTOR, v=V_CIRC*SPEED_FACTOR, r=URSCRIPT_BLEND)
  movel(apply_correction(p[-0.007599, 0.536545, 0.050005, 3.141576, 0.000000, 0.000000]), a=URSCRIPT_ACCEL*ACCEL_FACTOR, v=V_CIRC*SPEED_FACTOR, r=URSCRIPT_BLEND)
  movel(apply_correction(p[-0.001356, 0.539401, 0.050005, 3.141576, 0.000000, 0.000000]), a=URSCRIPT_ACCEL*ACCEL_FACTOR, v=V_CIRC*SPEED_FACTOR, r=URSCRIPT_BLEND)
  movel(apply_correction(p[-0.002041, 0.546340, 0.050005, 3.141576, 0.000000, 0.000000]), a=URSCRIPT_ACCEL*ACCEL_FACTOR, v=V_CIRC*SPEED_FACTOR, r=URSCRIPT_BLEND)
  movel(apply_correction(p[-0.008378, 0.549617, 0.050005, 3.141576, 0.000000, 0.000000]), a=URSCRIPT_ACCEL*ACCEL_FACTOR, v=V_CIRC*SPEED_FACTOR, r=URSCRIPT_BLEND)
  movel(apply_correction(p[-0.015100, 0.547118, 0.050005, 3.141576, 0.000000, 0.000000]), a=URSCRIPT_ACCEL*ACCEL_FACTOR, v=V_CIRC*SPEED_FACTOR, r=URSCRIPT_BLEND)
  movel(apply_correction(p[-0.017677, 0.540470, 0.050005, 3.141576, 0.000000, 0.000000]), a=URSCRIPT_ACCEL*ACCEL_FACTOR, v=V_CIRC*SPEED_FACTOR, r=URSCRIPT_BLEND)
  movel(apply_correction(p[-0.013312, 0.535048, 0.050005, 3.141576, 0.000000, 0.000000]), a=URSCRIPT_ACCEL*ACCEL_FACTOR, v=V_CIRC*SPEED_FACTOR, r=URSCRIPT_BLEND)
  movel(apply_correction(p[-0.006869, 0.537498, 0.050005, 3.141576, 0.000000, 0.000000]), a=URSCRIPT_ACCEL*ACCEL_FACTOR, v=V_CIRC*SPEED_FACTOR, r=URSCRIPT_BLEND)
  movel(apply_correction(p[-0.006196, 0.544557, 0.050005, 3.141576, 0.000000, 0.000000]), a=URSCRIPT_ACCEL*ACCEL_FACTOR, v=V_CIRC*SPEED_FACTOR, r=URSCRIPT_BLEND)
  movel(apply_correction(p[-0.011303, 0.549604, 0.050005, 3.141576, 0.000000, 0.000000]), a=URSCRIPT_ACCEL*ACCEL_FACTOR, v=V_CIRC*SPEED_FACTOR, r=URSCRIPT_BLEND)
  movel(apply_correction(p[-0.018457, 0.549307, 0.050005, 3.141576, 0.000000, 0.000000]), a=URSCRIPT_ACCEL*ACCEL_FACTOR, v=V_CIRC*SPEED_FACTOR, r=URSCRIPT_BLEND)
  movel(apply_correction(p[-0.022436, 0.543491, 0.050005, 3.141576, 0.000000, 0.000000]), a=URSCRIPT_ACCEL*ACCEL_FACTOR, v=V_CIRC*SPEED_FACTOR, r=URSCRIPT_BLEND)
  movel(apply_correction(p[-0.018669, 0.537715, 0.050005, 3.141576, 0.000000, 0.000000]), a=URSCRIPT_ACCEL*ACCEL_FACTOR, v=V_CIRC*SPEED_FACTOR, r=URSCRIPT_BLEND)
  movel(apply_correction(p[-0.011875, 0.539380, 0.050005, 3.141576, 0.000000, 0.000000]), a=URSCRIPT_ACCEL*ACCEL_FACTOR, v=V_CIRC*SPEED_FACTOR, r=URSCRIPT_BLEND)
  movel(apply_correction(p[-0.009742, 0.546188, 0.050005, 3.141576, 0.000000, 0.000000]), a=URSCRIPT_ACCEL*ACCEL_FACTOR, v=V_CIRC*SPEED_FACTOR, r=URSCRIPT_BLEND)
  movel(apply_correction(p[-0.013558, 0.552276, 0.050005, 3.141576, 0.000000, 0.000000]), a=URSCRIPT_ACCEL*ACCEL_FACTOR, v=V_CIRC*SPEED_FACTOR, r=URSCRIPT_BLEND)
  movel(apply_correction(p[-0.020613, 0.553566, 0.050005, 3.141576, 0.000000, 0.000000]), a=URSCRIPT_ACCEL*ACCEL_FACTOR, v=V_CIRC*SPEED_FACTOR, r=URSCRIPT_BLEND)
  movel(apply_correction(p[-0.025840, 0.548787, 0.050005, 3.141576, 0.000000, 0.000000]), a=URSCRIPT_ACCEL*ACCEL_FACTOR, v=V_CIRC*SPEED_FACTOR, r=URSCRIPT_BLEND)
  movel(apply_correction(p[-0.023792, 0.542172, 0.050005, 3.141576, 0.000000, 0.000000]), a=URSCRIPT_ACCEL*ACCEL_FACTOR, v=V_CIRC*SPEED_FACTOR, r=URSCRIPT_BLEND)
  movel(apply_correction(p[-0.016835, 0.542028, 0.050005, 3.141576, 0.000000, 0.000000]), a=URSCRIPT_ACCEL*ACCEL_FACTOR, v=V_CIRC*SPEED_FACTOR, r=URSCRIPT_BLEND)
  movel(apply_correction(p[-0.013339, 0.548221, 0.050005, 3.141576, 0.000000, 0.000000]), a=URSCRIPT_ACCEL*ACCEL_FACTOR, v=V_CIRC*SPEED_FACTOR, r=URSCRIPT_BLEND)
  movel(apply_correction(p[-0.015968, 0.554903, 0.050005, 3.141576, 0.000000, 0.000000]), a=URSCRIPT_ACCEL*ACCEL_FACTOR, v=V_CIRC*SPEED_FACTOR, r=URSCRIPT_BLEND)
  movel(apply_correction(p[-0.022664, 0.557493, 0.050005, 3.141576, 0.000000, 0.000000]), a=URSCRIPT_ACCEL*ACCEL_FACTOR, v=V_CIRC*SPEED_FACTOR, r=URSCRIPT_BLEND)
  movel(apply_correction(p[-0.028833, 0.553959, 0.050005, 3.141576, 0.000000, 0.000000]), a=URSCRIPT_ACCEL*ACCEL_FACTOR, v=V_CIRC*SPEED_FACTOR, r=URSCRIPT_BLEND)
  movel(apply_correction(p[-0.028635, 0.547007, 0.050005, 3.141576, 0.000000, 0.000000]), a=URSCRIPT_ACCEL*ACCEL_FACTOR, v=V_CIRC*SPEED_FACTOR, r=URSCRIPT_BLEND)
  movel(apply_correction(p[-0.022003, 0.545011, 0.050005, 3.141576, 0.000000, 0.000000]), a=URSCRIPT_ACCEL*ACCEL_FACTOR, v=V_CIRC*SPEED_FACTOR, r=URSCRIPT_BLEND)
  movel(apply_correction(p[-0.017259, 0.550270, 0.050005, 3.141576, 0.000000, 0.000000]), a=URSCRIPT_ACCEL*ACCEL_FACTOR, v=V_CIRC*SPEED_FACTOR, r=URSCRIPT_BLEND)
  movel(apply_correction(p[-0.018587, 0.557319, 0.050005, 3.141576, 0.000000, 0.000000]), a=URSCRIPT_ACCEL*ACCEL_FACTOR, v=V_CIRC*SPEED_FACTOR, r=URSCRIPT_BLEND)
  movel(apply_correction(p[-0.024697, 0.561102, 0.050005, 3.141576, 0.000000, 0.000000]), a=URSCRIPT_ACCEL*ACCEL_FACTOR, v=V_CIRC*SPEED_FACTOR, r=URSCRIPT_BLEND)
  movel(apply_correction(p[-0.031491, 0.558927, 0.050005, 3.141576, 0.000000, 0.000000]), a=URSCRIPT_ACCEL*ACCEL_FACTOR, v=V_CIRC*SPEED_FACTOR, r=URSCRIPT_BLEND)
  movel(apply_correction(p[-0.033105, 0.552122, 0.050005, 3.141576, 0.000000, 0.000000]), a=URSCRIPT_ACCEL*ACCEL_FACTOR, v=V_CIRC*SPEED_FACTOR, r=URSCRIPT_BLEND)
  movel(apply_correction(p[-0.027295, 0.548386, 0.050005, 3.141576, 0.000000, 0.000000]), a=URSCRIPT_ACCEL*ACCEL_FACTOR, v=V_CIRC*SPEED_FACTOR, r=URSCRIPT_BLEND)
  movel(apply_correction(p[-0.021500, 0.552402, 0.050005, 3.141576, 0.000000, 0.000000]), a=URSCRIPT_ACCEL*ACCEL_FACTOR, v=V_CIRC*SPEED_FACTOR, r=URSCRIPT_BLEND)
  movel(apply_correction(p[-0.021456, 0.559562, 0.050005, 3.141576, 0.000000, 0.000000]), a=URSCRIPT_ACCEL*ACCEL_FACTOR, v=V_CIRC*SPEED_FACTOR, r=URSCRIPT_BLEND)
  movel(apply_correction(p[-0.026772, 0.564399, 0.050005, 3.141576, 0.000000, 0.000000]), a=URSCRIPT_ACCEL*ACCEL_FACTOR, v=V_CIRC*SPEED_FACTOR, r=URSCRIPT_BLEND)
  movel(apply_correction(p[-0.033883, 0.563631, 0.050005, 3.141576, 0.000000, 0.000000]), a=URSCRIPT_ACCEL*ACCEL_FACTOR, v=V_CIRC*SPEED_FACTOR, r=URSCRIPT_BLEND)
  movel(apply_correction(p[-0.037145, 0.557401, 0.050005, 3.141576, 0.000000, 0.000000]), a=URSCRIPT_ACCEL*ACCEL_FACTOR, v=V_CIRC*SPEED_FACTOR, r=URSCRIPT_BLEND)
  movel(apply_correction(p[-0.032611, 0.552198, 0.050005, 3.141576, 0.000000, 0.000000]), a=URSCRIPT_ACCEL*ACCEL_FACTOR, v=V_CIRC*SPEED_FACTOR, r=URSCRIPT_BLEND)
  movel(apply_correction(p[-0.026054, 0.554687, 0.050005, 3.141576, 0.000000, 0.000000]), a=URSCRIPT_ACCEL*ACCEL_FACTOR, v=V_CIRC*SPEED_FACTOR, r=URSCRIPT_BLEND)
  movel(apply_correction(p[-0.024601, 0.561681, 0.050005, 3.141576, 0.000000, 0.000000]), a=URSCRIPT_ACCEL*ACCEL_FACTOR, v=V_CIRC*SPEED_FACTOR, r=URSCRIPT_BLEND)
  movel(apply_correction(p[-0.028946, 0.567405, 0.050004, 3.141576, 0.000000, 0.000000]), a=URSCRIPT_ACCEL*ACCEL_FACTOR, v=V_CIRC*SPEED_FACTOR, r=URSCRIPT_BLEND)
  movel(apply_correction(p[-0.036085, 0.568036, 0.050004, 3.141576, 0.000000, 0.000000]), a=URSCRIPT_ACCEL*ACCEL_FACTOR, v=V_CIRC*SPEED_FACTOR, r=URSCRIPT_BLEND)
  movel(apply_correction(p[-0.040740, 0.562720, 0.050005, 3.141576, 0.000000, 0.000000]), a=URSCRIPT_ACCEL*ACCEL_FACTOR, v=V_CIRC*SPEED_FACTOR, r=URSCRIPT_BLEND)
  movel(apply_correction(p[-0.037827, 0.556450, 0.050005, 3.141576, 0.000000, 0.000000]), a=URSCRIPT_ACCEL*ACCEL_FACTOR, v=V_CIRC*SPEED_FACTOR, r=URSCRIPT_BLEND)
  movel(apply_correction(p[-0.030891, 0.557198, 0.050005, 3.141576, 0.000000, 0.000000]), a=URSCRIPT_ACCEL*ACCEL_FACTOR, v=V_CIRC*SPEED_FACTOR, r=URSCRIPT_BLEND)
  movel(apply_correction(p[-0.028047, 0.563729, 0.050005, 3.141576, 0.000000, 0.000000]), a=URSCRIPT_ACCEL*ACCEL_FACTOR, v=V_CIRC*SPEED_FACTOR, r=URSCRIPT_BLEND)
  movel(apply_correction(p[-0.031268, 0.570149, 0.050004, 3.141576, 0.000000, 0.000000]), a=URSCRIPT_ACCEL*ACCEL_FACTOR, v=V_CIRC*SPEED_FACTOR, r=URSCRIPT_BLEND)
  movel(apply_correction(p[-0.038167, 0.572121, 0.050004, 3.141576, 0.000000, 0.000000]), a=URSCRIPT_ACCEL*ACCEL_FACTOR, v=V_CIRC*SPEED_FACTOR, r=URSCRIPT_BLEND)
  movel(apply_correction(p[-0.043920, 0.567963, 0.050004, 3.141576, 0.000000, 0.000000]), a=URSCRIPT_ACCEL*ACCEL_FACTOR, v=V_CIRC*SPEED_FACTOR, r=URSCRIPT_BLEND)
  movel(apply_correction(p[-0.042820, 0.561110, 0.050005, 3.141576, 0.000000, 0.000000]), a=URSCRIPT_ACCEL*ACCEL_FACTOR, v=V_CIRC*SPEED_FACTOR, r=URSCRIPT_BLEND)
  end_force_mode()
  movel(apply_correction(p[-0.042820, 0.561110, 0.060005, 3.141576, 0.000000, 0.000000]), a=URSCRIPT_ACCEL*ACCEL_FACTOR, v=0.2500*SPEED_FACTOR)
end

def cycle_2():
  # --- Cycle 2 - Circulaire (UI) ---
  movel(apply_correction(p[-0.032496, 0.557857, 0.060005, 3.141576, 0.000000, 0.000000]), a=URSCRIPT_ACCEL*ACCEL_FACTOR, v=0.2500*SPEED_FACTOR)
  sleep(0.2)
  zero_ftsensor()
  sleep(0.2)
  force_mode(MEAS_FRAME, [0, 0, 1, 0, 0, 0], [0, 0, -6.0, 0, 0, 0], 2, [0.008, 0.008, 0.04, 0.35, 0.35, 0.35])
  movel(apply_correction(p[-0.032496, 0.557857, 0.045005, 3.141576, 0.000000, 0.000000]), a=URSCRIPT_ACCEL*ACCEL_FACTOR, v=URSCRIPT_RECONTACT_V*SPEED_FACTOR)
  movel(apply_correction(p[-0.032496, 0.557857, 0.050005, 3.141576, 0.000000, 0.000000]), a=URSCRIPT_ACCEL*ACCEL_FACTOR, v=V_CIRC*SPEED_FACTOR, r=URSCRIPT_BLEND)
  movel(apply_correction(p[-0.029888, 0.564547, 0.050005, 3.141576, 0.000000, 0.000000]), a=URSCRIPT_ACCEL*ACCEL_FACTOR, v=V_CIRC*SPEED_FACTOR, r=URSCRIPT_BLEND)
  movel(apply_correction(p[-0.033403, 0.570730, 0.050004, 3.141576, 0.000000, 0.000000]), a=URSCRIPT_ACCEL*ACCEL_FACTOR, v=V_CIRC*SPEED_FACTOR, r=URSCRIPT_BLEND)
  movel(apply_correction(p[-0.040358, 0.570559, 0.050004, 3.141576, 0.000000, 0.000000]), a=URSCRIPT_ACCEL*ACCEL_FACTOR, v=V_CIRC*SPEED_FACTOR, r=URSCRIPT_BLEND)
  movel(apply_correction(p[-0.042379, 0.563934, 0.050005, 3.141576, 0.000000, 0.000000]), a=URSCRIPT_ACCEL*ACCEL_FACTOR, v=V_CIRC*SPEED_FACTOR, r=URSCRIPT_BLEND)
  movel(apply_correction(p[-0.037135, 0.559173, 0.050005, 3.141576, 0.000000, 0.000000]), a=URSCRIPT_ACCEL*ACCEL_FACTOR, v=V_CIRC*SPEED_FACTOR, r=URSCRIPT_BLEND)
  movel(apply_correction(p[-0.030084, 0.560482, 0.050005, 3.141576, 0.000000, 0.000000]), a=URSCRIPT_ACCEL*ACCEL_FACTOR, v=V_CIRC*SPEED_FACTOR, r=URSCRIPT_BLEND)
  movel(apply_correction(p[-0.026285, 0.566580, 0.050004, 3.141576, 0.000000, 0.000000]), a=URSCRIPT_ACCEL*ACCEL_FACTOR, v=V_CIRC*SPEED_FACTOR, r=URSCRIPT_BLEND)
  movel(apply_correction(p[-0.028440, 0.573381, 0.050004, 3.141576, 0.000000, 0.000000]), a=URSCRIPT_ACCEL*ACCEL_FACTOR, v=V_CIRC*SPEED_FACTOR, r=URSCRIPT_BLEND)
  movel(apply_correction(p[-0.035239, 0.575022, 0.050004, 3.141576, 0.000000, 0.000000]), a=URSCRIPT_ACCEL*ACCEL_FACTOR, v=V_CIRC*SPEED_FACTOR, r=URSCRIPT_BLEND)
  movel(apply_correction(p[-0.038997, 0.569228, 0.050004, 3.141576, 0.000000, 0.000000]), a=URSCRIPT_ACCEL*ACCEL_FACTOR, v=V_CIRC*SPEED_FACTOR, r=URSCRIPT_BLEND)
  movel(apply_correction(p[-0.035002, 0.563420, 0.050005, 3.141576, 0.000000, 0.000000]), a=URSCRIPT_ACCEL*ACCEL_FACTOR, v=V_CIRC*SPEED_FACTOR, r=URSCRIPT_BLEND)
  movel(apply_correction(p[-0.027843, 0.563354, 0.050005, 3.141576, 0.000000, 0.000000]), a=URSCRIPT_ACCEL*ACCEL_FACTOR, v=V_CIRC*SPEED_FACTOR, r=URSCRIPT_BLEND)
  movel(apply_correction(p[-0.022993, 0.568658, 0.050004, 3.141576, 0.000000, 0.000000]), a=URSCRIPT_ACCEL*ACCEL_FACTOR, v=V_CIRC*SPEED_FACTOR, r=URSCRIPT_BLEND)
  movel(apply_correction(p[-0.023740, 0.575771, 0.050004, 3.141576, 0.000000, 0.000000]), a=URSCRIPT_ACCEL*ACCEL_FACTOR, v=V_CIRC*SPEED_FACTOR, r=URSCRIPT_BLEND)
  movel(apply_correction(p[-0.029958, 0.579054, 0.050004, 3.141576, 0.000000, 0.000000]), a=URSCRIPT_ACCEL*ACCEL_FACTOR, v=V_CIRC*SPEED_FACTOR, r=URSCRIPT_BLEND)
  movel(apply_correction(p[-0.035180, 0.574542, 0.050004, 3.141576, 0.000000, 0.000000]), a=URSCRIPT_ACCEL*ACCEL_FACTOR, v=V_CIRC*SPEED_FACTOR, r=URSCRIPT_BLEND)
  movel(apply_correction(p[-0.032715, 0.567976, 0.050004, 3.141576, 0.000000, 0.000000]), a=URSCRIPT_ACCEL*ACCEL_FACTOR, v=V_CIRC*SPEED_FACTOR, r=URSCRIPT_BLEND)
  movel(apply_correction(p[-0.025725, 0.566502, 0.050004, 3.141576, 0.000000, 0.000000]), a=URSCRIPT_ACCEL*ACCEL_FACTOR, v=V_CIRC*SPEED_FACTOR, r=URSCRIPT_BLEND)
  movel(apply_correction(p[-0.019989, 0.570833, 0.050004, 3.141576, 0.000000, 0.000000]), a=URSCRIPT_ACCEL*ACCEL_FACTOR, v=V_CIRC*SPEED_FACTOR, r=URSCRIPT_BLEND)
  movel(apply_correction(p[-0.019339, 0.577970, 0.050004, 3.141576, 0.000000, 0.000000]), a=URSCRIPT_ACCEL*ACCEL_FACTOR, v=V_CIRC*SPEED_FACTOR, r=URSCRIPT_BLEND)
  movel(apply_correction(p[-0.024640, 0.582644, 0.050004, 3.141576, 0.000000, 0.000000]), a=URSCRIPT_ACCEL*ACCEL_FACTOR, v=V_CIRC*SPEED_FACTOR, r=URSCRIPT_BLEND)
  movel(apply_correction(p[-0.030921, 0.579756, 0.050004, 3.141576, 0.000000, 0.000000]), a=URSCRIPT_ACCEL*ACCEL_FACTOR, v=V_CIRC*SPEED_FACTOR, r=URSCRIPT_BLEND)
  movel(apply_correction(p[-0.030201, 0.572817, 0.050004, 3.141576, 0.000000, 0.000000]), a=URSCRIPT_ACCEL*ACCEL_FACTOR, v=V_CIRC*SPEED_FACTOR, r=URSCRIPT_BLEND)
  movel(apply_correction(p[-0.023678, 0.569955, 0.050004, 3.141576, 0.000000, 0.000000]), a=URSCRIPT_ACCEL*ACCEL_FACTOR, v=V_CIRC*SPEED_FACTOR, r=URSCRIPT_BLEND)
  movel(apply_correction(p[-0.017249, 0.573156, 0.050004, 3.141576, 0.000000, 0.000000]), a=URSCRIPT_ACCEL*ACCEL_FACTOR, v=V_CIRC*SPEED_FACTOR, r=URSCRIPT_BLEND)
  movel(apply_correction(p[-0.015259, 0.580051, 0.050004, 3.141576, 0.000000, 0.000000]), a=URSCRIPT_ACCEL*ACCEL_FACTOR, v=V_CIRC*SPEED_FACTOR, r=URSCRIPT_BLEND)
  movel(apply_correction(p[-0.019398, 0.585817, 0.050004, 3.141576, 0.000000, 0.000000]), a=URSCRIPT_ACCEL*ACCEL_FACTOR, v=V_CIRC*SPEED_FACTOR, r=URSCRIPT_BLEND)
  movel(apply_correction(p[-0.026254, 0.584744, 0.050004, 3.141576, 0.000000, 0.000000]), a=URSCRIPT_ACCEL*ACCEL_FACTOR, v=V_CIRC*SPEED_FACTOR, r=URSCRIPT_BLEND)
  movel(apply_correction(p[-0.027384, 0.577897, 0.050004, 3.141576, 0.000000, 0.000000]), a=URSCRIPT_ACCEL*ACCEL_FACTOR, v=V_CIRC*SPEED_FACTOR, r=URSCRIPT_BLEND)
  movel(apply_correction(p[-0.021645, 0.573721, 0.050004, 3.141576, 0.000000, 0.000000]), a=URSCRIPT_ACCEL*ACCEL_FACTOR, v=V_CIRC*SPEED_FACTOR, r=URSCRIPT_BLEND)
  movel(apply_correction(p[-0.014740, 0.575673, 0.050004, 3.141576, 0.000000, 0.000000]), a=URSCRIPT_ACCEL*ACCEL_FACTOR, v=V_CIRC*SPEED_FACTOR, r=URSCRIPT_BLEND)
  movel(apply_correction(p[-0.011501, 0.582084, 0.050004, 3.141576, 0.000000, 0.000000]), a=URSCRIPT_ACCEL*ACCEL_FACTOR, v=V_CIRC*SPEED_FACTOR, r=URSCRIPT_BLEND)
  movel(apply_correction(p[-0.014326, 0.588624, 0.050004, 3.141576, 0.000000, 0.000000]), a=URSCRIPT_ACCEL*ACCEL_FACTOR, v=V_CIRC*SPEED_FACTOR, r=URSCRIPT_BLEND)
  movel(apply_correction(p[-0.021257, 0.589399, 0.050004, 3.141576, 0.000000, 0.000000]), a=URSCRIPT_ACCEL*ACCEL_FACTOR, v=V_CIRC*SPEED_FACTOR, r=URSCRIPT_BLEND)
  movel(apply_correction(p[-0.024200, 0.583141, 0.050004, 3.141576, 0.000000, 0.000000]), a=URSCRIPT_ACCEL*ACCEL_FACTOR, v=V_CIRC*SPEED_FACTOR, r=URSCRIPT_BLEND)
  movel(apply_correction(p[-0.019560, 0.577812, 0.050004, 3.141576, 0.000000, 0.000000]), a=URSCRIPT_ACCEL*ACCEL_FACTOR, v=V_CIRC*SPEED_FACTOR, r=URSCRIPT_BLEND)
  movel(apply_correction(p[-0.012421, 0.578421, 0.050004, 3.141576, 0.000000, 0.000000]), a=URSCRIPT_ACCEL*ACCEL_FACTOR, v=V_CIRC*SPEED_FACTOR, r=URSCRIPT_BLEND)
  movel(apply_correction(p[-0.008061, 0.584133, 0.050004, 3.141576, 0.000000, 0.000000]), a=URSCRIPT_ACCEL*ACCEL_FACTOR, v=V_CIRC*SPEED_FACTOR, r=URSCRIPT_BLEND)
  movel(apply_correction(p[-0.009521, 0.591120, 0.050004, 3.141576, 0.000000, 0.000000]), a=URSCRIPT_ACCEL*ACCEL_FACTOR, v=V_CIRC*SPEED_FACTOR, r=URSCRIPT_BLEND)
  movel(apply_correction(p[-0.016085, 0.593389, 0.050004, 3.141576, 0.000000, 0.000000]), a=URSCRIPT_ACCEL*ACCEL_FACTOR, v=V_CIRC*SPEED_FACTOR, r=URSCRIPT_BLEND)
  movel(apply_correction(p[-0.020236, 0.587906, 0.050004, 3.141576, 0.000000, 0.000000]), a=URSCRIPT_ACCEL*ACCEL_FACTOR, v=V_CIRC*SPEED_FACTOR, r=URSCRIPT_BLEND)
  movel(apply_correction(p[-0.017032, 0.581581, 0.050004, 3.141576, 0.000000, 0.000000]), a=URSCRIPT_ACCEL*ACCEL_FACTOR, v=V_CIRC*SPEED_FACTOR, r=URSCRIPT_BLEND)
  movel(apply_correction(p[-0.009998, 0.580074, 0.050004, 3.141576, 0.000000, 0.000000]), a=URSCRIPT_ACCEL*ACCEL_FACTOR, v=V_CIRC*SPEED_FACTOR, r=URSCRIPT_BLEND)
  movel(apply_correction(p[-0.004123, 0.584197, 0.050004, 3.141576, 0.000000, 0.000000]), a=URSCRIPT_ACCEL*ACCEL_FACTOR, v=V_CIRC*SPEED_FACTOR, r=URSCRIPT_BLEND)
  movel(apply_correction(p[-0.003908, 0.591243, 0.050004, 3.141576, 0.000000, 0.000000]), a=URSCRIPT_ACCEL*ACCEL_FACTOR, v=V_CIRC*SPEED_FACTOR, r=URSCRIPT_BLEND)
  movel(apply_correction(p[-0.010173, 0.594044, 0.050004, 3.141576, 0.000000, 0.000000]), a=URSCRIPT_ACCEL*ACCEL_FACTOR, v=V_CIRC*SPEED_FACTOR, r=URSCRIPT_BLEND)
  movel(apply_correction(p[-0.015011, 0.588994, 0.050004, 3.141576, 0.000000, 0.000000]), a=URSCRIPT_ACCEL*ACCEL_FACTOR, v=V_CIRC*SPEED_FACTOR, r=URSCRIPT_BLEND)
  movel(apply_correction(p[-0.013519, 0.582011, 0.050004, 3.141576, 0.000000, 0.000000]), a=URSCRIPT_ACCEL*ACCEL_FACTOR, v=V_CIRC*SPEED_FACTOR, r=URSCRIPT_BLEND)
  movel(apply_correction(p[-0.007341, 0.578371, 0.050004, 3.141576, 0.000000, 0.000000]), a=URSCRIPT_ACCEL*ACCEL_FACTOR, v=V_CIRC*SPEED_FACTOR, r=URSCRIPT_BLEND)
  movel(apply_correction(p[-0.000583, 0.580621, 0.050004, 3.141576, 0.000000, 0.000000]), a=URSCRIPT_ACCEL*ACCEL_FACTOR, v=V_CIRC*SPEED_FACTOR, r=URSCRIPT_BLEND)
  movel(apply_correction(p[0.000654, 0.587459, 0.050004, 3.141576, 0.000000, 0.000000]), a=URSCRIPT_ACCEL*ACCEL_FACTOR, v=V_CIRC*SPEED_FACTOR, r=URSCRIPT_BLEND)
  movel(apply_correction(p[-0.005450, 0.590705, 0.050004, 3.141576, 0.000000, 0.000000]), a=URSCRIPT_ACCEL*ACCEL_FACTOR, v=V_CIRC*SPEED_FACTOR, r=URSCRIPT_BLEND)
  movel(apply_correction(p[-0.011313, 0.586692, 0.050004, 3.141576, 0.000000, 0.000000]), a=URSCRIPT_ACCEL*ACCEL_FACTOR, v=V_CIRC*SPEED_FACTOR, r=URSCRIPT_BLEND)
  movel(apply_correction(p[-0.012006, 0.579542, 0.050004, 3.141576, 0.000000, 0.000000]), a=URSCRIPT_ACCEL*ACCEL_FACTOR, v=V_CIRC*SPEED_FACTOR, r=URSCRIPT_BLEND)
  movel(apply_correction(p[-0.007247, 0.574197, 0.050004, 3.141576, 0.000000, 0.000000]), a=URSCRIPT_ACCEL*ACCEL_FACTOR, v=V_CIRC*SPEED_FACTOR, r=URSCRIPT_BLEND)
  movel(apply_correction(p[-0.000249, 0.574916, 0.050004, 3.141576, 0.000000, 0.000000]), a=URSCRIPT_ACCEL*ACCEL_FACTOR, v=V_CIRC*SPEED_FACTOR, r=URSCRIPT_BLEND)
  movel(apply_correction(p[0.001510, 0.581584, 0.050004, 3.141576, 0.000000, 0.000000]), a=URSCRIPT_ACCEL*ACCEL_FACTOR, v=V_CIRC*SPEED_FACTOR, r=URSCRIPT_BLEND)
  movel(apply_correction(p[-0.004223, 0.585659, 0.050004, 3.141576, 0.000000, 0.000000]), a=URSCRIPT_ACCEL*ACCEL_FACTOR, v=V_CIRC*SPEED_FACTOR, r=URSCRIPT_BLEND)
  movel(apply_correction(p[-0.010995, 0.583363, 0.050004, 3.141576, 0.000000, 0.000000]), a=URSCRIPT_ACCEL*ACCEL_FACTOR, v=V_CIRC*SPEED_FACTOR, r=URSCRIPT_BLEND)
  movel(apply_correction(p[-0.013924, 0.576811, 0.050004, 3.141576, 0.000000, 0.000000]), a=URSCRIPT_ACCEL*ACCEL_FACTOR, v=V_CIRC*SPEED_FACTOR, r=URSCRIPT_BLEND)
  movel(apply_correction(p[-0.010852, 0.570399, 0.050004, 3.141576, 0.000000, 0.000000]), a=URSCRIPT_ACCEL*ACCEL_FACTOR, v=V_CIRC*SPEED_FACTOR, r=URSCRIPT_BLEND)
  movel(apply_correction(p[-0.003894, 0.569992, 0.050004, 3.141576, 0.000000, 0.000000]), a=URSCRIPT_ACCEL*ACCEL_FACTOR, v=V_CIRC*SPEED_FACTOR, r=URSCRIPT_BLEND)
  movel(apply_correction(p[-0.001310, 0.576409, 0.050004, 3.141576, 0.000000, 0.000000]), a=URSCRIPT_ACCEL*ACCEL_FACTOR, v=V_CIRC*SPEED_FACTOR, r=URSCRIPT_BLEND)
  movel(apply_correction(p[-0.006194, 0.581525, 0.050004, 3.141576, 0.000000, 0.000000]), a=URSCRIPT_ACCEL*ACCEL_FACTOR, v=V_CIRC*SPEED_FACTOR, r=URSCRIPT_BLEND)
  movel(apply_correction(p[-0.013307, 0.580639, 0.050004, 3.141576, 0.000000, 0.000000]), a=URSCRIPT_ACCEL*ACCEL_FACTOR, v=V_CIRC*SPEED_FACTOR, r=URSCRIPT_BLEND)
  movel(apply_correction(p[-0.017454, 0.574769, 0.050004, 3.141576, 0.000000, 0.000000]), a=URSCRIPT_ACCEL*ACCEL_FACTOR, v=V_CIRC*SPEED_FACTOR, r=URSCRIPT_BLEND)
  movel(apply_correction(p[-0.015738, 0.567838, 0.050004, 3.141576, 0.000000, 0.000000]), a=URSCRIPT_ACCEL*ACCEL_FACTOR, v=V_CIRC*SPEED_FACTOR, r=URSCRIPT_BLEND)
  movel(apply_correction(p[-0.009079, 0.565660, 0.050004, 3.141576, 0.000000, 0.000000]), a=URSCRIPT_ACCEL*ACCEL_FACTOR, v=V_CIRC*SPEED_FACTOR, r=URSCRIPT_BLEND)
  movel(apply_correction(p[-0.004826, 0.571096, 0.050004, 3.141576, 0.000000, 0.000000]), a=URSCRIPT_ACCEL*ACCEL_FACTOR, v=V_CIRC*SPEED_FACTOR, r=URSCRIPT_BLEND)
  movel(apply_correction(p[-0.008367, 0.577178, 0.050004, 3.141576, 0.000000, 0.000000]), a=URSCRIPT_ACCEL*ACCEL_FACTOR, v=V_CIRC*SPEED_FACTOR, r=URSCRIPT_BLEND)
  movel(apply_correction(p[-0.015504, 0.577683, 0.050004, 3.141576, 0.000000, 0.000000]), a=URSCRIPT_ACCEL*ACCEL_FACTOR, v=V_CIRC*SPEED_FACTOR, r=URSCRIPT_BLEND)
  movel(apply_correction(p[-0.020652, 0.572667, 0.050004, 3.141576, 0.000000, 0.000000]), a=URSCRIPT_ACCEL*ACCEL_FACTOR, v=V_CIRC*SPEED_FACTOR, r=URSCRIPT_BLEND)
  movel(apply_correction(p[-0.020346, 0.565518, 0.050004, 3.141576, 0.000000, 0.000000]), a=URSCRIPT_ACCEL*ACCEL_FACTOR, v=V_CIRC*SPEED_FACTOR, r=URSCRIPT_BLEND)
  movel(apply_correction(p[-0.014385, 0.561767, 0.050005, 3.141576, 0.000000, 0.000000]), a=URSCRIPT_ACCEL*ACCEL_FACTOR, v=V_CIRC*SPEED_FACTOR, r=URSCRIPT_BLEND)
  movel(apply_correction(p[-0.008782, 0.565800, 0.050004, 3.141576, 0.000000, 0.000000]), a=URSCRIPT_ACCEL*ACCEL_FACTOR, v=V_CIRC*SPEED_FACTOR, r=URSCRIPT_BLEND)
  movel(apply_correction(p[-0.010719, 0.572527, 0.050004, 3.141576, 0.000000, 0.000000]), a=URSCRIPT_ACCEL*ACCEL_FACTOR, v=V_CIRC*SPEED_FACTOR, r=URSCRIPT_BLEND)
  movel(apply_correction(p[-0.017594, 0.574443, 0.050004, 3.141576, 0.000000, 0.000000]), a=URSCRIPT_ACCEL*ACCEL_FACTOR, v=V_CIRC*SPEED_FACTOR, r=URSCRIPT_BLEND)
  movel(apply_correction(p[-0.023570, 0.570450, 0.050004, 3.141576, 0.000000, 0.000000]), a=URSCRIPT_ACCEL*ACCEL_FACTOR, v=V_CIRC*SPEED_FACTOR, r=URSCRIPT_BLEND)
  movel(apply_correction(p[-0.024648, 0.563362, 0.050005, 3.141576, 0.000000, 0.000000]), a=URSCRIPT_ACCEL*ACCEL_FACTOR, v=V_CIRC*SPEED_FACTOR, r=URSCRIPT_BLEND)
  movel(apply_correction(p[-0.019690, 0.558311, 0.050005, 3.141576, 0.000000, 0.000000]), a=URSCRIPT_ACCEL*ACCEL_FACTOR, v=V_CIRC*SPEED_FACTOR, r=URSCRIPT_BLEND)
  movel(apply_correction(p[-0.013173, 0.560644, 0.050005, 3.141576, 0.000000, 0.000000]), a=URSCRIPT_ACCEL*ACCEL_FACTOR, v=V_CIRC*SPEED_FACTOR, r=URSCRIPT_BLEND)
  movel(apply_correction(p[-0.013320, 0.567606, 0.050004, 3.141576, 0.000000, 0.000000]), a=URSCRIPT_ACCEL*ACCEL_FACTOR, v=V_CIRC*SPEED_FACTOR, r=URSCRIPT_BLEND)
  movel(apply_correction(p[-0.019631, 0.570894, 0.050004, 3.141576, 0.000000, 0.000000]), a=URSCRIPT_ACCEL*ACCEL_FACTOR, v=V_CIRC*SPEED_FACTOR, r=URSCRIPT_BLEND)
  movel(apply_correction(p[-0.026235, 0.568072, 0.050004, 3.141576, 0.000000, 0.000000]), a=URSCRIPT_ACCEL*ACCEL_FACTOR, v=V_CIRC*SPEED_FACTOR, r=URSCRIPT_BLEND)
  movel(apply_correction(p[-0.028627, 0.561302, 0.050005, 3.141576, 0.000000, 0.000000]), a=URSCRIPT_ACCEL*ACCEL_FACTOR, v=V_CIRC*SPEED_FACTOR, r=URSCRIPT_BLEND)
  movel(apply_correction(p[-0.024888, 0.555260, 0.050005, 3.141576, 0.000000, 0.000000]), a=URSCRIPT_ACCEL*ACCEL_FACTOR, v=V_CIRC*SPEED_FACTOR, r=URSCRIPT_BLEND)
  movel(apply_correction(p[-0.017954, 0.555751, 0.050005, 3.141576, 0.000000, 0.000000]), a=URSCRIPT_ACCEL*ACCEL_FACTOR, v=V_CIRC*SPEED_FACTOR, r=URSCRIPT_BLEND)
  movel(apply_correction(p[-0.016245, 0.562467, 0.050005, 3.141576, 0.000000, 0.000000]), a=URSCRIPT_ACCEL*ACCEL_FACTOR, v=V_CIRC*SPEED_FACTOR, r=URSCRIPT_BLEND)
  movel(apply_correction(p[-0.021689, 0.567014, 0.050004, 3.141576, 0.000000, 0.000000]), a=URSCRIPT_ACCEL*ACCEL_FACTOR, v=V_CIRC*SPEED_FACTOR, r=URSCRIPT_BLEND)
  movel(apply_correction(p[-0.028641, 0.565300, 0.050005, 3.141576, 0.000000, 0.000000]), a=URSCRIPT_ACCEL*ACCEL_FACTOR, v=V_CIRC*SPEED_FACTOR, r=URSCRIPT_BLEND)
  movel(apply_correction(p[-0.031974, 0.558949, 0.050005, 3.141576, 0.000000, 0.000000]), a=URSCRIPT_ACCEL*ACCEL_FACTOR, v=V_CIRC*SPEED_FACTOR, r=URSCRIPT_BLEND)
  movel(apply_correction(p[-0.029410, 0.552284, 0.050005, 3.141576, 0.000000, 0.000000]), a=URSCRIPT_ACCEL*ACCEL_FACTOR, v=V_CIRC*SPEED_FACTOR, r=URSCRIPT_BLEND)
  movel(apply_correction(p[-0.022597, 0.550409, 0.050005, 3.141576, 0.000000, 0.000000]), a=URSCRIPT_ACCEL*ACCEL_FACTOR, v=V_CIRC*SPEED_FACTOR, r=URSCRIPT_BLEND)
  movel(apply_correction(p[-0.018007, 0.555612, 0.050005, 3.141576, 0.000000, 0.000000]), a=URSCRIPT_ACCEL*ACCEL_FACTOR, v=V_CIRC*SPEED_FACTOR, r=URSCRIPT_BLEND)
  movel(apply_correction(p[-0.021445, 0.561607, 0.050005, 3.141576, 0.000000, 0.000000]), a=URSCRIPT_ACCEL*ACCEL_FACTOR, v=V_CIRC*SPEED_FACTOR, r=URSCRIPT_BLEND)
  movel(apply_correction(p[-0.028444, 0.560907, 0.050005, 3.141576, 0.000000, 0.000000]), a=URSCRIPT_ACCEL*ACCEL_FACTOR, v=V_CIRC*SPEED_FACTOR, r=URSCRIPT_BLEND)
  movel(apply_correction(p[-0.031888, 0.554670, 0.050005, 3.141576, 0.000000, 0.000000]), a=URSCRIPT_ACCEL*ACCEL_FACTOR, v=V_CIRC*SPEED_FACTOR, r=URSCRIPT_BLEND)
  movel(apply_correction(p[-0.029404, 0.547959, 0.050005, 3.141576, 0.000000, 0.000000]), a=URSCRIPT_ACCEL*ACCEL_FACTOR, v=V_CIRC*SPEED_FACTOR, r=URSCRIPT_BLEND)
  movel(apply_correction(p[-0.022754, 0.545340, 0.050005, 3.141576, 0.000000, 0.000000]), a=URSCRIPT_ACCEL*ACCEL_FACTOR, v=V_CIRC*SPEED_FACTOR, r=URSCRIPT_BLEND)
  movel(apply_correction(p[-0.016650, 0.548949, 0.050005, 3.141576, 0.000000, 0.000000]), a=URSCRIPT_ACCEL*ACCEL_FACTOR, v=V_CIRC*SPEED_FACTOR, r=URSCRIPT_BLEND)
  movel(apply_correction(p[-0.016888, 0.555928, 0.050005, 3.141576, 0.000000, 0.000000]), a=URSCRIPT_ACCEL*ACCEL_FACTOR, v=V_CIRC*SPEED_FACTOR, r=URSCRIPT_BLEND)
  movel(apply_correction(p[-0.023497, 0.558002, 0.050005, 3.141576, 0.000000, 0.000000]), a=URSCRIPT_ACCEL*ACCEL_FACTOR, v=V_CIRC*SPEED_FACTOR, r=URSCRIPT_BLEND)
  movel(apply_correction(p[-0.027927, 0.552554, 0.050005, 3.141576, 0.000000, 0.000000]), a=URSCRIPT_ACCEL*ACCEL_FACTOR, v=V_CIRC*SPEED_FACTOR, r=URSCRIPT_BLEND)
  movel(apply_correction(p[-0.025735, 0.545775, 0.050005, 3.141576, 0.000000, 0.000000]), a=URSCRIPT_ACCEL*ACCEL_FACTOR, v=V_CIRC*SPEED_FACTOR, r=URSCRIPT_BLEND)
  movel(apply_correction(p[-0.019062, 0.543110, 0.050005, 3.141576, 0.000000, 0.000000]), a=URSCRIPT_ACCEL*ACCEL_FACTOR, v=V_CIRC*SPEED_FACTOR, r=URSCRIPT_BLEND)
  movel(apply_correction(p[-0.012631, 0.546307, 0.050005, 3.141576, 0.000000, 0.000000]), a=URSCRIPT_ACCEL*ACCEL_FACTOR, v=V_CIRC*SPEED_FACTOR, r=URSCRIPT_BLEND)
  movel(apply_correction(p[-0.011081, 0.553247, 0.050005, 3.141576, 0.000000, 0.000000]), a=URSCRIPT_ACCEL*ACCEL_FACTOR, v=V_CIRC*SPEED_FACTOR, r=URSCRIPT_BLEND)
  movel(apply_correction(p[-0.016101, 0.558111, 0.050005, 3.141576, 0.000000, 0.000000]), a=URSCRIPT_ACCEL*ACCEL_FACTOR, v=V_CIRC*SPEED_FACTOR, r=URSCRIPT_BLEND)
  movel(apply_correction(p[-0.022343, 0.555169, 0.050005, 3.141576, 0.000000, 0.000000]), a=URSCRIPT_ACCEL*ACCEL_FACTOR, v=V_CIRC*SPEED_FACTOR, r=URSCRIPT_BLEND)
  movel(apply_correction(p[-0.021751, 0.548196, 0.050005, 3.141576, 0.000000, 0.000000]), a=URSCRIPT_ACCEL*ACCEL_FACTOR, v=V_CIRC*SPEED_FACTOR, r=URSCRIPT_BLEND)
  movel(apply_correction(p[-0.015311, 0.545149, 0.050005, 3.141576, 0.000000, 0.000000]), a=URSCRIPT_ACCEL*ACCEL_FACTOR, v=V_CIRC*SPEED_FACTOR, r=URSCRIPT_BLEND)
  movel(apply_correction(p[-0.008807, 0.548200, 0.050005, 3.141576, 0.000000, 0.000000]), a=URSCRIPT_ACCEL*ACCEL_FACTOR, v=V_CIRC*SPEED_FACTOR, r=URSCRIPT_BLEND)
  movel(apply_correction(p[-0.006651, 0.555046, 0.050005, 3.141576, 0.000000, 0.000000]), a=URSCRIPT_ACCEL*ACCEL_FACTOR, v=V_CIRC*SPEED_FACTOR, r=URSCRIPT_BLEND)
  movel(apply_correction(p[-0.010629, 0.560928, 0.050005, 3.141576, 0.000000, 0.000000]), a=URSCRIPT_ACCEL*ACCEL_FACTOR, v=V_CIRC*SPEED_FACTOR, r=URSCRIPT_BLEND)
  movel(apply_correction(p[-0.017524, 0.560094, 0.050005, 3.141576, 0.000000, 0.000000]), a=URSCRIPT_ACCEL*ACCEL_FACTOR, v=V_CIRC*SPEED_FACTOR, r=URSCRIPT_BLEND)
  movel(apply_correction(p[-0.018888, 0.553294, 0.050005, 3.141576, 0.000000, 0.000000]), a=URSCRIPT_ACCEL*ACCEL_FACTOR, v=V_CIRC*SPEED_FACTOR, r=URSCRIPT_BLEND)
  movel(apply_correction(p[-0.013273, 0.548960, 0.050005, 3.141576, 0.000000, 0.000000]), a=URSCRIPT_ACCEL*ACCEL_FACTOR, v=V_CIRC*SPEED_FACTOR, r=URSCRIPT_BLEND)
  movel(apply_correction(p[-0.006323, 0.550743, 0.050005, 3.141576, 0.000000, 0.000000]), a=URSCRIPT_ACCEL*ACCEL_FACTOR, v=V_CIRC*SPEED_FACTOR, r=URSCRIPT_BLEND)
  movel(apply_correction(p[-0.002935, 0.557077, 0.050005, 3.141576, 0.000000, 0.000000]), a=URSCRIPT_ACCEL*ACCEL_FACTOR, v=V_CIRC*SPEED_FACTOR, r=URSCRIPT_BLEND)
  movel(apply_correction(p[-0.005584, 0.563693, 0.050005, 3.141576, 0.000000, 0.000000]), a=URSCRIPT_ACCEL*ACCEL_FACTOR, v=V_CIRC*SPEED_FACTOR, r=URSCRIPT_BLEND)
  movel(apply_correction(p[-0.012491, 0.564699, 0.050005, 3.141576, 0.000000, 0.000000]), a=URSCRIPT_ACCEL*ACCEL_FACTOR, v=V_CIRC*SPEED_FACTOR, r=URSCRIPT_BLEND)
  movel(apply_correction(p[-0.015653, 0.558553, 0.050005, 3.141576, 0.000000, 0.000000]), a=URSCRIPT_ACCEL*ACCEL_FACTOR, v=V_CIRC*SPEED_FACTOR, r=URSCRIPT_BLEND)
  movel(apply_correction(p[-0.011179, 0.553089, 0.050005, 3.141576, 0.000000, 0.000000]), a=URSCRIPT_ACCEL*ACCEL_FACTOR, v=V_CIRC*SPEED_FACTOR, r=URSCRIPT_BLEND)
  movel(apply_correction(p[-0.004027, 0.553523, 0.050005, 3.141576, 0.000000, 0.000000]), a=URSCRIPT_ACCEL*ACCEL_FACTOR, v=V_CIRC*SPEED_FACTOR, r=URSCRIPT_BLEND)
  movel(apply_correction(p[0.000468, 0.559132, 0.050005, 3.141576, 0.000000, 0.000000]), a=URSCRIPT_ACCEL*ACCEL_FACTOR, v=V_CIRC*SPEED_FACTOR, r=URSCRIPT_BLEND)
  movel(apply_correction(p[-0.000784, 0.566169, 0.050004, 3.141576, 0.000000, 0.000000]), a=URSCRIPT_ACCEL*ACCEL_FACTOR, v=V_CIRC*SPEED_FACTOR, r=URSCRIPT_BLEND)
  movel(apply_correction(p[-0.007254, 0.568889, 0.050004, 3.141576, 0.000000, 0.000000]), a=URSCRIPT_ACCEL*ACCEL_FACTOR, v=V_CIRC*SPEED_FACTOR, r=URSCRIPT_BLEND)
  movel(apply_correction(p[-0.011995, 0.563874, 0.050005, 3.141576, 0.000000, 0.000000]), a=URSCRIPT_ACCEL*ACCEL_FACTOR, v=V_CIRC*SPEED_FACTOR, r=URSCRIPT_BLEND)
  movel(apply_correction(p[-0.008954, 0.557539, 0.050005, 3.141576, 0.000000, 0.000000]), a=URSCRIPT_ACCEL*ACCEL_FACTOR, v=V_CIRC*SPEED_FACTOR, r=URSCRIPT_BLEND)
  movel(apply_correction(p[-0.001870, 0.556571, 0.050005, 3.141576, 0.000000, 0.000000]), a=URSCRIPT_ACCEL*ACCEL_FACTOR, v=V_CIRC*SPEED_FACTOR, r=URSCRIPT_BLEND)
  movel(apply_correction(p[0.003570, 0.561266, 0.050005, 3.141576, 0.000000, 0.000000]), a=URSCRIPT_ACCEL*ACCEL_FACTOR, v=V_CIRC*SPEED_FACTOR, r=URSCRIPT_BLEND)
  movel(apply_correction(p[0.003725, 0.568426, 0.050004, 3.141576, 0.000000, 0.000000]), a=URSCRIPT_ACCEL*ACCEL_FACTOR, v=V_CIRC*SPEED_FACTOR, r=URSCRIPT_BLEND)
  movel(apply_correction(p[-0.001936, 0.572638, 0.050004, 3.141576, 0.000000, 0.000000]), a=URSCRIPT_ACCEL*ACCEL_FACTOR, v=V_CIRC*SPEED_FACTOR, r=URSCRIPT_BLEND)
  movel(apply_correction(p[-0.007892, 0.569138, 0.050004, 3.141576, 0.000000, 0.000000]), a=URSCRIPT_ACCEL*ACCEL_FACTOR, v=V_CIRC*SPEED_FACTOR, r=URSCRIPT_BLEND)
  movel(apply_correction(p[-0.006528, 0.562284, 0.050005, 3.141576, 0.000000, 0.000000]), a=URSCRIPT_ACCEL*ACCEL_FACTOR, v=V_CIRC*SPEED_FACTOR, r=URSCRIPT_BLEND)
  movel(apply_correction(p[0.000196, 0.559909, 0.050005, 3.141576, 0.000000, 0.000000]), a=URSCRIPT_ACCEL*ACCEL_FACTOR, v=V_CIRC*SPEED_FACTOR, r=URSCRIPT_BLEND)
  movel(apply_correction(p[0.006401, 0.563532, 0.050005, 3.141576, 0.000000, 0.000000]), a=URSCRIPT_ACCEL*ACCEL_FACTOR, v=V_CIRC*SPEED_FACTOR, r=URSCRIPT_BLEND)
  movel(apply_correction(p[0.007921, 0.570542, 0.050004, 3.141576, 0.000000, 0.000000]), a=URSCRIPT_ACCEL*ACCEL_FACTOR, v=V_CIRC*SPEED_FACTOR, r=URSCRIPT_BLEND)
  movel(apply_correction(p[0.003329, 0.575913, 0.050004, 3.141576, 0.000000, 0.000000]), a=URSCRIPT_ACCEL*ACCEL_FACTOR, v=V_CIRC*SPEED_FACTOR, r=URSCRIPT_BLEND)
  movel(apply_correction(p[-0.003298, 0.574095, 0.050004, 3.141576, 0.000000, 0.000000]), a=URSCRIPT_ACCEL*ACCEL_FACTOR, v=V_CIRC*SPEED_FACTOR, r=URSCRIPT_BLEND)
  movel(apply_correction(p[-0.003661, 0.567148, 0.050004, 3.141576, 0.000000, 0.000000]), a=URSCRIPT_ACCEL*ACCEL_FACTOR, v=V_CIRC*SPEED_FACTOR, r=URSCRIPT_BLEND)
  movel(apply_correction(p[0.002239, 0.563147, 0.050005, 3.141576, 0.000000, 0.000000]), a=URSCRIPT_ACCEL*ACCEL_FACTOR, v=V_CIRC*SPEED_FACTOR, r=URSCRIPT_BLEND)
  movel(apply_correction(p[0.009196, 0.564880, 0.050005, 3.141576, 0.000000, 0.000000]), a=URSCRIPT_ACCEL*ACCEL_FACTOR, v=V_CIRC*SPEED_FACTOR, r=URSCRIPT_BLEND)
  movel(apply_correction(p[0.012546, 0.571174, 0.050004, 3.141576, 0.000000, 0.000000]), a=URSCRIPT_ACCEL*ACCEL_FACTOR, v=V_CIRC*SPEED_FACTOR, r=URSCRIPT_BLEND)
  movel(apply_correction(p[0.009051, 0.577193, 0.050004, 3.141576, 0.000000, 0.000000]), a=URSCRIPT_ACCEL*ACCEL_FACTOR, v=V_CIRC*SPEED_FACTOR, r=URSCRIPT_BLEND)
  movel(apply_correction(p[0.002326, 0.575811, 0.050004, 3.141576, 0.000000, 0.000000]), a=URSCRIPT_ACCEL*ACCEL_FACTOR, v=V_CIRC*SPEED_FACTOR, r=URSCRIPT_BLEND)
  movel(apply_correction(p[0.000722, 0.568917, 0.050004, 3.141576, 0.000000, 0.000000]), a=URSCRIPT_ACCEL*ACCEL_FACTOR, v=V_CIRC*SPEED_FACTOR, r=URSCRIPT_BLEND)
  movel(apply_correction(p[0.005225, 0.563313, 0.050005, 3.141576, 0.000000, 0.000000]), a=URSCRIPT_ACCEL*ACCEL_FACTOR, v=V_CIRC*SPEED_FACTOR, r=URSCRIPT_BLEND)
  movel(apply_correction(p[0.012386, 0.562788, 0.050005, 3.141576, 0.000000, 0.000000]), a=URSCRIPT_ACCEL*ACCEL_FACTOR, v=V_CIRC*SPEED_FACTOR, r=URSCRIPT_BLEND)
  movel(apply_correction(p[0.017100, 0.568047, 0.050004, 3.141576, 0.000000, 0.000000]), a=URSCRIPT_ACCEL*ACCEL_FACTOR, v=V_CIRC*SPEED_FACTOR, r=URSCRIPT_BLEND)
  movel(apply_correction(p[0.014245, 0.574289, 0.050004, 3.141576, 0.000000, 0.000000]), a=URSCRIPT_ACCEL*ACCEL_FACTOR, v=V_CIRC*SPEED_FACTOR, r=URSCRIPT_BLEND)
  movel(apply_correction(p[0.007306, 0.573605, 0.050004, 3.141576, 0.000000, 0.000000]), a=URSCRIPT_ACCEL*ACCEL_FACTOR, v=V_CIRC*SPEED_FACTOR, r=URSCRIPT_BLEND)
  movel(apply_correction(p[0.004029, 0.567268, 0.050004, 3.141576, 0.000000, 0.000000]), a=URSCRIPT_ACCEL*ACCEL_FACTOR, v=V_CIRC*SPEED_FACTOR, r=URSCRIPT_BLEND)
  movel(apply_correction(p[0.006528, 0.560546, 0.050005, 3.141576, 0.000000, 0.000000]), a=URSCRIPT_ACCEL*ACCEL_FACTOR, v=V_CIRC*SPEED_FACTOR, r=URSCRIPT_BLEND)
  movel(apply_correction(p[0.013176, 0.557969, 0.050005, 3.141576, 0.000000, 0.000000]), a=URSCRIPT_ACCEL*ACCEL_FACTOR, v=V_CIRC*SPEED_FACTOR, r=URSCRIPT_BLEND)
  movel(apply_correction(p[0.018597, 0.562334, 0.050005, 3.141576, 0.000000, 0.000000]), a=URSCRIPT_ACCEL*ACCEL_FACTOR, v=V_CIRC*SPEED_FACTOR, r=URSCRIPT_BLEND)
  movel(apply_correction(p[0.016147, 0.568777, 0.050004, 3.141576, 0.000000, 0.000000]), a=URSCRIPT_ACCEL*ACCEL_FACTOR, v=V_CIRC*SPEED_FACTOR, r=URSCRIPT_BLEND)
  movel(apply_correction(p[0.009089, 0.569450, 0.050004, 3.141576, 0.000000, 0.000000]), a=URSCRIPT_ACCEL*ACCEL_FACTOR, v=V_CIRC*SPEED_FACTOR, r=URSCRIPT_BLEND)
  movel(apply_correction(p[0.004042, 0.564343, 0.050005, 3.141576, 0.000000, 0.000000]), a=URSCRIPT_ACCEL*ACCEL_FACTOR, v=V_CIRC*SPEED_FACTOR, r=URSCRIPT_BLEND)
  movel(apply_correction(p[0.004339, 0.557189, 0.050005, 3.141576, 0.000000, 0.000000]), a=URSCRIPT_ACCEL*ACCEL_FACTOR, v=V_CIRC*SPEED_FACTOR, r=URSCRIPT_BLEND)
  movel(apply_correction(p[0.010155, 0.553210, 0.050005, 3.141576, 0.000000, 0.000000]), a=URSCRIPT_ACCEL*ACCEL_FACTOR, v=V_CIRC*SPEED_FACTOR, r=URSCRIPT_BLEND)
  movel(apply_correction(p[0.015931, 0.556976, 0.050005, 3.141576, 0.000000, 0.000000]), a=URSCRIPT_ACCEL*ACCEL_FACTOR, v=V_CIRC*SPEED_FACTOR, r=URSCRIPT_BLEND)
  movel(apply_correction(p[0.014266, 0.563771, 0.050005, 3.141576, 0.000000, 0.000000]), a=URSCRIPT_ACCEL*ACCEL_FACTOR, v=V_CIRC*SPEED_FACTOR, r=URSCRIPT_BLEND)
  movel(apply_correction(p[0.007458, 0.565904, 0.050004, 3.141576, 0.000000, 0.000000]), a=URSCRIPT_ACCEL*ACCEL_FACTOR, v=V_CIRC*SPEED_FACTOR, r=URSCRIPT_BLEND)
  movel(apply_correction(p[0.001370, 0.562087, 0.050005, 3.141576, 0.000000, 0.000000]), a=URSCRIPT_ACCEL*ACCEL_FACTOR, v=V_CIRC*SPEED_FACTOR, r=URSCRIPT_BLEND)
  movel(apply_correction(p[0.000080, 0.555033, 0.050005, 3.141576, 0.000000, 0.000000]), a=URSCRIPT_ACCEL*ACCEL_FACTOR, v=V_CIRC*SPEED_FACTOR, r=URSCRIPT_BLEND)
  movel(apply_correction(p[0.004858, 0.549806, 0.050005, 3.141576, 0.000000, 0.000000]), a=URSCRIPT_ACCEL*ACCEL_FACTOR, v=V_CIRC*SPEED_FACTOR, r=URSCRIPT_BLEND)
  movel(apply_correction(p[0.011474, 0.551853, 0.050005, 3.141576, 0.000000, 0.000000]), a=URSCRIPT_ACCEL*ACCEL_FACTOR, v=V_CIRC*SPEED_FACTOR, r=URSCRIPT_BLEND)
  movel(apply_correction(p[0.011618, 0.558811, 0.050005, 3.141576, 0.000000, 0.000000]), a=URSCRIPT_ACCEL*ACCEL_FACTOR, v=V_CIRC*SPEED_FACTOR, r=URSCRIPT_BLEND)
  movel(apply_correction(p[0.005425, 0.562307, 0.050005, 3.141576, 0.000000, 0.000000]), a=URSCRIPT_ACCEL*ACCEL_FACTOR, v=V_CIRC*SPEED_FACTOR, r=URSCRIPT_BLEND)
  movel(apply_correction(p[-0.001257, 0.559678, 0.050005, 3.141576, 0.000000, 0.000000]), a=URSCRIPT_ACCEL*ACCEL_FACTOR, v=V_CIRC*SPEED_FACTOR, r=URSCRIPT_BLEND)
  movel(apply_correction(p[-0.003848, 0.552982, 0.050005, 3.141576, 0.000000, 0.000000]), a=URSCRIPT_ACCEL*ACCEL_FACTOR, v=V_CIRC*SPEED_FACTOR, r=URSCRIPT_BLEND)
  movel(apply_correction(p[-0.000313, 0.546813, 0.050005, 3.141576, 0.000000, 0.000000]), a=URSCRIPT_ACCEL*ACCEL_FACTOR, v=V_CIRC*SPEED_FACTOR, r=URSCRIPT_BLEND)
  movel(apply_correction(p[0.006639, 0.547011, 0.050005, 3.141576, 0.000000, 0.000000]), a=URSCRIPT_ACCEL*ACCEL_FACTOR, v=V_CIRC*SPEED_FACTOR, r=URSCRIPT_BLEND)
  movel(apply_correction(p[0.008635, 0.553643, 0.050005, 3.141576, 0.000000, 0.000000]), a=URSCRIPT_ACCEL*ACCEL_FACTOR, v=V_CIRC*SPEED_FACTOR, r=URSCRIPT_BLEND)
  movel(apply_correction(p[0.003375, 0.558386, 0.050005, 3.141576, 0.000000, 0.000000]), a=URSCRIPT_ACCEL*ACCEL_FACTOR, v=V_CIRC*SPEED_FACTOR, r=URSCRIPT_BLEND)
  movel(apply_correction(p[-0.003673, 0.557058, 0.050005, 3.141576, 0.000000, 0.000000]), a=URSCRIPT_ACCEL*ACCEL_FACTOR, v=V_CIRC*SPEED_FACTOR, r=URSCRIPT_BLEND)
  movel(apply_correction(p[-0.007456, 0.550949, 0.050005, 3.141576, 0.000000, 0.000000]), a=URSCRIPT_ACCEL*ACCEL_FACTOR, v=V_CIRC*SPEED_FACTOR, r=URSCRIPT_BLEND)
  movel(apply_correction(p[-0.005281, 0.544155, 0.050005, 3.141576, 0.000000, 0.000000]), a=URSCRIPT_ACCEL*ACCEL_FACTOR, v=V_CIRC*SPEED_FACTOR, r=URSCRIPT_BLEND)
  movel(apply_correction(p[0.001524, 0.542541, 0.050005, 3.141576, 0.000000, 0.000000]), a=URSCRIPT_ACCEL*ACCEL_FACTOR, v=V_CIRC*SPEED_FACTOR, r=URSCRIPT_BLEND)
  movel(apply_correction(p[0.005260, 0.548350, 0.050005, 3.141576, 0.000000, 0.000000]), a=URSCRIPT_ACCEL*ACCEL_FACTOR, v=V_CIRC*SPEED_FACTOR, r=URSCRIPT_BLEND)
  movel(apply_correction(p[0.001244, 0.554146, 0.050005, 3.141576, 0.000000, 0.000000]), a=URSCRIPT_ACCEL*ACCEL_FACTOR, v=V_CIRC*SPEED_FACTOR, r=URSCRIPT_BLEND)
  movel(apply_correction(p[-0.005917, 0.554190, 0.050005, 3.141576, 0.000000, 0.000000]), a=URSCRIPT_ACCEL*ACCEL_FACTOR, v=V_CIRC*SPEED_FACTOR, r=URSCRIPT_BLEND)
  movel(apply_correction(p[-0.010753, 0.548874, 0.050005, 3.141576, 0.000000, 0.000000]), a=URSCRIPT_ACCEL*ACCEL_FACTOR, v=V_CIRC*SPEED_FACTOR, r=URSCRIPT_BLEND)
  movel(apply_correction(p[-0.009985, 0.541763, 0.050005, 3.141576, 0.000000, 0.000000]), a=URSCRIPT_ACCEL*ACCEL_FACTOR, v=V_CIRC*SPEED_FACTOR, r=URSCRIPT_BLEND)
  movel(apply_correction(p[-0.003756, 0.538500, 0.050005, 3.141576, 0.000000, 0.000000]), a=URSCRIPT_ACCEL*ACCEL_FACTOR, v=V_CIRC*SPEED_FACTOR, r=URSCRIPT_BLEND)
  movel(apply_correction(p[0.001448, 0.543035, 0.050005, 3.141576, 0.000000, 0.000000]), a=URSCRIPT_ACCEL*ACCEL_FACTOR, v=V_CIRC*SPEED_FACTOR, r=URSCRIPT_BLEND)
  movel(apply_correction(p[-0.001042, 0.549592, 0.050005, 3.141576, 0.000000, 0.000000]), a=URSCRIPT_ACCEL*ACCEL_FACTOR, v=V_CIRC*SPEED_FACTOR, r=URSCRIPT_BLEND)
  movel(apply_correction(p[-0.008035, 0.551044, 0.050005, 3.141576, 0.000000, 0.000000]), a=URSCRIPT_ACCEL*ACCEL_FACTOR, v=V_CIRC*SPEED_FACTOR, r=URSCRIPT_BLEND)
  movel(apply_correction(p[-0.013760, 0.546700, 0.050005, 3.141576, 0.000000, 0.000000]), a=URSCRIPT_ACCEL*ACCEL_FACTOR, v=V_CIRC*SPEED_FACTOR, r=URSCRIPT_BLEND)
  movel(apply_correction(p[-0.014391, 0.539561, 0.050005, 3.141576, 0.000000, 0.000000]), a=URSCRIPT_ACCEL*ACCEL_FACTOR, v=V_CIRC*SPEED_FACTOR, r=URSCRIPT_BLEND)
  movel(apply_correction(p[-0.009075, 0.534905, 0.050005, 3.141576, 0.000000, 0.000000]), a=URSCRIPT_ACCEL*ACCEL_FACTOR, v=V_CIRC*SPEED_FACTOR, r=URSCRIPT_BLEND)
  movel(apply_correction(p[-0.002804, 0.537819, 0.050005, 3.141576, 0.000000, 0.000000]), a=URSCRIPT_ACCEL*ACCEL_FACTOR, v=V_CIRC*SPEED_FACTOR, r=URSCRIPT_BLEND)
  movel(apply_correction(p[-0.003553, 0.544755, 0.050005, 3.141576, 0.000000, 0.000000]), a=URSCRIPT_ACCEL*ACCEL_FACTOR, v=V_CIRC*SPEED_FACTOR, r=URSCRIPT_BLEND)
  movel(apply_correction(p[-0.010084, 0.547599, 0.050005, 3.141576, 0.000000, 0.000000]), a=URSCRIPT_ACCEL*ACCEL_FACTOR, v=V_CIRC*SPEED_FACTOR, r=URSCRIPT_BLEND)
  movel(apply_correction(p[-0.016503, 0.544378, 0.050005, 3.141576, 0.000000, 0.000000]), a=URSCRIPT_ACCEL*ACCEL_FACTOR, v=V_CIRC*SPEED_FACTOR, r=URSCRIPT_BLEND)
  movel(apply_correction(p[-0.018476, 0.537479, 0.050005, 3.141576, 0.000000, 0.000000]), a=URSCRIPT_ACCEL*ACCEL_FACTOR, v=V_CIRC*SPEED_FACTOR, r=URSCRIPT_BLEND)
  movel(apply_correction(p[-0.014318, 0.531726, 0.050005, 3.141576, 0.000000, 0.000000]), a=URSCRIPT_ACCEL*ACCEL_FACTOR, v=V_CIRC*SPEED_FACTOR, r=URSCRIPT_BLEND)
  movel(apply_correction(p[-0.007464, 0.532826, 0.050005, 3.141576, 0.000000, 0.000000]), a=URSCRIPT_ACCEL*ACCEL_FACTOR, v=V_CIRC*SPEED_FACTOR, r=URSCRIPT_BLEND)
  end_force_mode()
  movel(apply_correction(p[-0.007464, 0.532826, 0.060005, 3.141576, 0.000000, 0.000000]), a=URSCRIPT_ACCEL*ACCEL_FACTOR, v=0.2500*SPEED_FACTOR)
end

